LIN {X 0,Y 409.415,Z 604.793,A -85,B 0,C 180,E1 19415.298,E2 19415.298} C_VEL
LIN {X 0,Y 409.395,Z 604.8,A -85,B 0,C 180,E1 19411.55,E2 19411.55} C_VEL
LIN {X 0,Y 409.394,Z 604.798,A -85,B 0,C 180,E1 19407.666,E2 19407.666} C_VEL
LIN {X 0,Y 409.417,Z 604.797,A -85,B 0,C 180,E1 19403.936,E2 19403.936} C_VEL
LIN {X 0,Y 409.444,Z 604.799,A -85,B 0,C 180,E1 19400.041,E2 19400.041} C_VEL
LIN {X 0,Y 409.442,Z 604.791,A -85,B 0,C 180,E1 19396.087,E2 19396.087} C_VEL
LIN {X 0,Y 409.455,Z 604.99,A -85,B 0,C 180,E1 19392.185,E2 19392.185} C_VEL
LIN {X 0,Y 416.656,Z 624.819,A -85,B 0,C 180,E1 19389.076,E2 19389.076} C_VEL
LIN {X 0,Y 424.364,Z 647.273,A -85,B 0,C 180,E1 19385.922,E2 19385.922} C_VEL
LIN {X 0,Y 424.911,Z 649.682,A -85,B 0,C 180,E1 19385.62,E2 19385.62} C_VEL
LIN {X 0,Y 420.58,Z 693.435,A -85,B 0,C 180,E1 19381.336,E2 19381.336} C_VEL
LIN {X 0,Y 423.293,Z 718.927,A -85,B 0,C 180,E1 19380.669,E2 19380.669} C_VEL
LIN {X 0,Y 420.432,Z 893.062,A -85,B 0,C 180,E1 19377.697,E2 19377.697} C_VEL
LIN {X 0,Y 419.51,Z 911.823,A -85,B 0,C 180,E1 19377.138,E2 19377.138} C_VEL
LIN {X 0,Y 418.324,Z 929.671,A -85,B 0,C 180,E1 19376.358,E2 19376.358} C_VEL
LIN {X 0,Y 416.943,Z 947.056,A -85,B 0,C 180,E1 19375.337,E2 19375.337} C_VEL
LIN {X 0,Y 415.337,Z 964.706,A -85,B 0,C 180,E1 19374.007,E2 19374.007} C_VEL
LIN {X 0,Y 413.794,Z 980.489,A -85,B 0,C 180,E1 19372.525,E2 19372.525} C_VEL
LIN {X 0,Y 412.341,Z 995.458,A -85,B 0,C 180,E1 19370.808,E2 19370.808} C_VEL
LIN {X 0,Y 411.026,Z 1009.443,A -85,B 0,C 180,E1 19368.866,E2 19368.866} C_VEL
LIN {X 0,Y 409.929,Z 1022.117,A -85,B 0,C 180,E1 19366.727,E2 19366.727} C_VEL
LIN {X 0,Y 409.153,Z 1033.229,A -85,B 0,C 180,E1 19364.434,E2 19364.434} C_VEL
LIN {X 0,Y 408.687,Z 1042.25,A -85,B 0,C 180,E1 19362.146,E2 19362.146} C_VEL
LIN {X 0,Y 408.488,Z 1049.838,A -85,B 0,C 180,E1 19359.724,E2 19359.724} C_VEL
LIN {X 0,Y 408.479,Z 1055.589,A -85,B 0,C 180,E1 19357.313,E2 19357.313} C_VEL
LIN {X 0,Y 408.559,Z 1059.642,A -85,B 0,C 180,E1 19354.914,E2 19354.914} C_VEL
LIN {X 0,Y 408.661,Z 1062.08,A -85,B 0,C 180,E1 19352.524,E2 19352.524} C_VEL
LIN {X 0,Y 408.725,Z 1062.933,A -85,B 0,C 180,E1 19350,E2 19350} C_VEL
LIN {X 0,Y 408.668,Z 1062.03,A -85,B 0,C 180,E1 19347.476,E2 19347.476} C_VEL
LIN {X 0,Y 408.564,Z 1059.37,A -85,B 0,C 180,E1 19344.946,E2 19344.946} C_VEL
LIN {X 0,Y 408.484,Z 1054.907,A -85,B 0,C 180,E1 19342.405,E2 19342.405} C_VEL
LIN {X 0,Y 408.514,Z 1048.531,A -85,B 0,C 180,E1 19339.85,E2 19339.85} C_VEL
LIN {X 0,Y 408.758,Z 1040.58,A -85,B 0,C 180,E1 19337.419,E2 19337.419} C_VEL
LIN {X 0,Y 409.269,Z 1031.268,A -85,B 0,C 180,E1 19335.137,E2 19335.137} C_VEL
LIN {X 0,Y 410.115,Z 1019.776,A -85,B 0,C 180,E1 19332.843,E2 19332.843} C_VEL
LIN {X 0,Y 411.249,Z 1007.148,A -85,B 0,C 180,E1 19330.765,E2 19330.765} C_VEL
LIN {X 0,Y 412.638,Z 992.973,A -85,B 0,C 180,E1 19328.836,E2 19328.836} C_VEL
LIN {X 0,Y 414.238,Z 977.091,A -85,B 0,C 180,E1 19327.057,E2 19327.057} C_VEL
LIN {X 0,Y 415.901,Z 960.831,A -85,B 0,C 180,E1 19325.575,E2 19325.575} C_VEL
LIN {X 0,Y 417.509,Z 943.547,A -85,B 0,C 180,E1 19324.313,E2 19324.313} C_VEL
LIN {X 0,Y 418.963,Z 925.915,A -85,B 0,C 180,E1 19323.315,E2 19323.315} C_VEL
LIN {X 0,Y 420.212,Z 907.373,A -85,B 0,C 180,E1 19322.551,E2 19322.551} C_VEL
LIN {X 0,Y 421.062,Z 888.73,A -85,B 0,C 180,E1 19322.043,E2 19322.043} C_VEL
LIN {X 0,Y 423.931,Z 716.146,A -85,B 0,C 180,E1 19319.049,E2 19319.049} C_VEL
LIN {X 0,Y 421.384,Z 693.883,A -85,B 0,C 180,E1 19318.403,E2 19318.403} C_VEL
LIN {X 0,Y 426.24,Z 650.86,A -85,B 0,C 180,E1 19314.066,E2 19314.066} C_VEL
LIN {X 0,Y 421.233,Z 635.297,A -85,B 0,C 180,E1 19311.719,E2 19311.719} C_VEL
LIN {X 0,Y 415.789,Z 620.626,A -85,B 0,C 180,E1 19309.243,E2 19309.243} C_VEL
LIN {X 0,Y 410.723,Z 608.35,A -85,B 0,C 180,E1 19306.913,E2 19306.913} C_VEL
LIN {X 0,Y 409.462,Z 604.966,A -85,B 0,C 180,E1 19306.185,E2 19306.185} C_VEL
LIN {X 0,Y 409.409,Z 604.798,A -85,B 0,C 180,E1 19302.38,E2 19302.38} C_VEL
LIN {X 0,Y 409.385,Z 604.791,A -85,B 0,C 180,E1 19298.7,E2 19298.7} C_VEL
LIN {X 0,Y 409.392,Z 604.791,A -85,B 0,C 180,E1 19294.854,E2 19294.854} C_VEL
LIN {X 0,Y 409.423,Z 604.786,A -85,B 0,C 180,E1 19291.18,E2 19291.18} C_VEL
LIN {X 0,Y 409.443,Z 604.781,A -85,B 0,C 180,E1 19287.329,E2 19287.329} C_VEL
LIN {X 0,Y 409.427,Z 604.781,A -85,B 0,C 180,E1 19283.457,E2 19283.457} C_VEL
LIN {X 0,Y 409.402,Z 604.787,A -85,B 0,C 180,E1 19279.696,E2 19279.696} C_VEL
LIN {X 0,Y 409.395,Z 604.797,A -85,B 0,C 180,E1 19275.875,E2 19275.875} C_VEL
LIN {X 0,Y 409.4,Z 604.801,A -85,B 0,C 180,E1 19271.981,E2 19271.981} C_VEL
LIN {X 0,Y 409.417,Z 604.789,A -85,B 0,C 180,E1 19268.143,E2 19268.143} C_VEL
LIN {X 0,Y 409.435,Z 604.778,A -85,B 0,C 180,E1 19264.341,E2 19264.341} C_VEL
LIN {X 0,Y 409.443,Z 604.781,A -85,B 0,C 180,E1 19260.419,E2 19260.419} C_VEL
LIN {X 0,Y 409.424,Z 604.794,A -85,B 0,C 180,E1 19256.499,E2 19256.499} C_VEL
LIN {X 0,Y 409.408,Z 604.799,A -85,B 0,C 180,E1 19252.704,E2 19252.704} C_VEL
LIN {X 0,Y 409.407,Z 604.8,A -85,B 0,C 180,E1 19248.733,E2 19248.733} C_VEL
LIN {X 0,Y 409.408,Z 604.801,A -85,B 0,C 180,E1 19244.725,E2 19244.725} C_VEL
LIN {X 0,Y 409.421,Z 604.8,A -85,B 0,C 180,E1 19240.898,E2 19240.898} C_VEL
LIN {X 0,Y 409.439,Z 604.792,A -85,B 0,C 180,E1 19237,E2 19237} C_VEL
LIN {X 0,Y 409.445,Z 604.787,A -85,B 0,C 180,E1 19232.986,E2 19232.986} C_VEL
LIN {X 0,Y 409.477,Z 605.015,A -85,B 0,C 180,E1 19229.195,E2 19229.195} C_VEL
LIN {X 0,Y 414.075,Z 618.311,A -85,B 0,C 180,E1 19226.096,E2 19226.096} C_VEL
LIN {X 0,Y 418.411,Z 632.268,A -85,B 0,C 180,E1 19223.144,E2 19223.144} C_VEL
LIN {X 0,Y 421.571,Z 644.812,A -85,B 0,C 180,E1 19220.709,E2 19220.709} C_VEL
LIN {X 0,Y 418.574,Z 672.307,A -85,B 0,C 180,E1 19216.567,E2 19216.567} C_VEL
LIN {X 0,Y 415.962,Z 700.171,A -85,B 0,C 180,E1 19212.443,E2 19212.443} C_VEL
LIN {X 0,Y 415.414,Z 707.768,A -85,B 0,C 180,E1 19211.384,E2 19211.384} C_VEL
LIN {X 0,Y 420.157,Z 732.939,A -85,B 0,C 180,E1 19210.505,E2 19210.505} C_VEL
LIN {X 0,Y 418.107,Z 830.68,A -85,B 0,C 180,E1 19208.658,E2 19208.658} C_VEL
LIN {X 0,Y 417.55,Z 846.98,A -85,B 0,C 180,E1 19208.08,E2 19208.08} C_VEL
LIN {X 0,Y 416.769,Z 861.253,A -85,B 0,C 180,E1 19207.317,E2 19207.317} C_VEL
LIN {X 0,Y 415.733,Z 875.611,A -85,B 0,C 180,E1 19206.274,E2 19206.274} C_VEL
LIN {X 0,Y 414.577,Z 888.557,A -85,B 0,C 180,E1 19205.029,E2 19205.029} C_VEL
LIN {X 0,Y 413.441,Z 900.019,A -85,B 0,C 180,E1 19203.629,E2 19203.629} C_VEL
LIN {X 0,Y 412.248,Z 911.043,A -85,B 0,C 180,E1 19201.909,E2 19201.909} C_VEL
LIN {X 0,Y 411.279,Z 919.508,A -85,B 0,C 180,E1 19200.214,E2 19200.214} C_VEL
LIN {X 0,Y 410.461,Z 926.728,A -85,B 0,C 180,E1 19198.36,E2 19198.36} C_VEL
LIN {X 0,Y 409.834,Z 932.478,A -85,B 0,C 180,E1 19196.36,E2 19196.36} C_VEL
LIN {X 0,Y 409.412,Z 936.698,A -85,B 0,C 180,E1 19194.223,E2 19194.223} C_VEL
LIN {X 0,Y 409.166,Z 939.127,A -85,B 0,C 180,E1 19191.955,E2 19191.955} C_VEL
LIN {X 0,Y 409.084,Z 939.659,A -85,B 0,C 180,E1 19189.779,E2 19189.779} C_VEL
LIN {X 0,Y 409.082,Z 939.537,A -85,B 0,C 180,E1 19189.241,E2 19189.241} C_VEL
LIN {X 0,Y 408.111,Z 939.093,A -85,B 0,C 180,E1 19188.162,E2 19188.162} C_VEL
LIN {X 0,Y 403.994,Z 937.675,A -85,B 0,C 180,E1 19186.285,E2 19186.285} C_VEL
LIN {X 0,Y 401.746,Z 935.756,A -85,B 0,C 180,E1 19184.919,E2 19184.919} C_VEL
LIN {X 0,Y 401.569,Z 934.669,A -85,B 0,C 180,E1 19184.384,E2 19184.384} C_VEL
LIN {X 0,Y 402.038,Z 929.349,A -85,B 0,C 180,E1 19182.35,E2 19182.35} C_VEL
LIN {X 0,Y 402.753,Z 921.963,A -85,B 0,C 180,E1 19180.296,E2 19180.296} C_VEL
LIN {X 0,Y 403.589,Z 913.727,A -85,B 0,C 180,E1 19178.548,E2 19178.548} C_VEL
LIN {X 0,Y 404.638,Z 903.344,A -85,B 0,C 180,E1 19176.812,E2 19176.812} C_VEL
LIN {X 0,Y 405.741,Z 891.203,A -85,B 0,C 180,E1 19175.231,E2 19175.231} C_VEL
LIN {X 0,Y 406.821,Z 878.561,A -85,B 0,C 180,E1 19173.946,E2 19173.946} C_VEL
LIN {X 0,Y 407.794,Z 865.03,A -85,B 0,C 180,E1 19172.881,E2 19172.881} C_VEL
LIN {X 0,Y 408.6,Z 850.501,A -85,B 0,C 180,E1 19172.033,E2 19172.033} C_VEL
LIN {X 0,Y 409.183,Z 835.057,A -85,B 0,C 180,E1 19171.41,E2 19171.41} C_VEL
LIN {X 0,Y 409.575,Z 814.247,A -85,B 0,C 180,E1 19170.942,E2 19170.942} C_VEL
LIN {X 0,Y 410.942,Z 731.935,A -85,B 0,C 180,E1 19169.426,E2 19169.426} C_VEL
LIN {X 0,Y 406.656,Z 707.352,A -85,B 0,C 180,E1 19168.661,E2 19168.661} C_VEL
LIN {X 0,Y 409.009,Z 677.997,A -85,B 0,C 180,E1 19164.388,E2 19164.388} C_VEL
LIN {X 0,Y 411.552,Z 650.681,A -85,B 0,C 180,E1 19160.349,E2 19160.349} C_VEL
LIN {X 0,Y 412.189,Z 643.268,A -85,B 0,C 180,E1 19159.235,E2 19159.235} C_VEL
LIN {X 0,Y 407.405,Z 625.4,A -85,B 0,C 180,E1 19155.938,E2 19155.938} C_VEL
LIN {X 0,Y 402.302,Z 608.499,A -85,B 0,C 180,E1 19152.627,E2 19152.627} C_VEL
LIN {X 0,Y 401.507,Z 605.885,A -85,B 0,C 180,E1 19152.013,E2 19152.013} C_VEL
LIN {X 0,Y 401.5,Z 605.772,A -85,B 0,C 180,E1 19148.065,E2 19148.065} C_VEL
LIN {X 0,Y 401.498,Z 605.771,A -85,B 0,C 180,E1 19144.004,E2 19144.004} C_VEL
LIN {X 0,Y 401.499,Z 605.737,A -85,B 0,C 180,E1 19140.07,E2 19140.07} C_VEL
LIN {X 0,Y 401.502,Z 605.778,A -85,B 0,C 180,E1 19136.024,E2 19136.024} C_VEL
LIN {X 0,Y 401.502,Z 605.772,A -85,B 0,C 180,E1 19132.04,E2 19132.04} C_VEL
LIN {X 0,Y 401.498,Z 605.772,A -85,B 0,C 180,E1 19128.126,E2 19128.126} C_VEL
LIN {X 0,Y 401.491,Z 605.787,A -85,B 0,C 180,E1 19124.173,E2 19124.173} C_VEL
LIN {X 0,Y 401.477,Z 605.762,A -85,B 0,C 180,E1 19120.351,E2 19120.351} C_VEL
LIN {X 0,Y 401.478,Z 605.785,A -85,B 0,C 180,E1 19116.351,E2 19116.351} C_VEL
LIN {X 0,Y 401.479,Z 605.771,A -85,B 0,C 180,E1 19112.374,E2 19112.374} C_VEL
LIN {X 0,Y 401.495,Z 605.778,A -85,B 0,C 180,E1 19108.466,E2 19108.466} C_VEL
LIN {X 0,Y 401.499,Z 605.765,A -85,B 0,C 180,E1 19104.575,E2 19104.575} C_VEL
LIN {X 0,Y 401.506,Z 605.779,A -85,B 0,C 180,E1 19100.709,E2 19100.709} C_VEL
LIN {X 0,Y 401.492,Z 605.755,A -85,B 0,C 180,E1 19096.791,E2 19096.791} C_VEL
LIN {X 0,Y 401.476,Z 605.789,A -85,B 0,C 180,E1 19092.953,E2 19092.953} C_VEL
LIN {X 0,Y 401.464,Z 605.755,A -85,B 0,C 180,E1 19089.028,E2 19089.028} C_VEL
LIN {X 0,Y 401.468,Z 605.784,A -85,B 0,C 180,E1 19085.144,E2 19085.144} C_VEL
LIN {X 0,Y 401.474,Z 605.759,A -85,B 0,C 180,E1 19081.285,E2 19081.285} C_VEL
LIN {X 0,Y 401.495,Z 605.783,A -85,B 0,C 180,E1 19077.431,E2 19077.431} C_VEL
LIN {X 0,Y 401.509,Z 605.756,A -85,B 0,C 180,E1 19073.423,E2 19073.423} C_VEL
LIN {X 0,Y 401.503,Z 605.786,A -85,B 0,C 180,E1 19069.381,E2 19069.381} C_VEL
LIN {X 0,Y 401.501,Z 605.762,A -85,B 0,C 180,E1 19065.433,E2 19065.433} C_VEL
LIN {X 0,Y 401.477,Z 605.788,A -85,B 0,C 180,E1 19061.562,E2 19061.562} C_VEL
LIN {X 0,Y 401.453,Z 605.782,A -85,B 0,C 180,E1 19057.755,E2 19057.755} C_VEL
LIN {X 0,Y 401.456,Z 605.772,A -85,B 0,C 180,E1 19053.843,E2 19053.843} C_VEL
LIN {X 0,Y 401.471,Z 605.781,A -85,B 0,C 180,E1 19050.077,E2 19050.077} C_VEL
LIN {X 0,Y 401.494,Z 605.781,A -85,B 0,C 180,E1 19046.266,E2 19046.266} C_VEL
LIN {X 0,Y 401.506,Z 605.78,A -85,B 0,C 180,E1 19042.365,E2 19042.365} C_VEL
LIN {X 0,Y 401.484,Z 605.78,A -85,B 0,C 180,E1 19038.513,E2 19038.513} C_VEL
LIN {X 0,Y 401.455,Z 605.786,A -85,B 0,C 180,E1 19034.78,E2 19034.78} C_VEL
LIN {X 0,Y 401.487,Z 606.048,A -85,B 0,C 180,E1 19032.879,E2 19032.879} C_VEL
LIN {X 0,Y 408.321,Z 624.696,A -85,B 0,C 180,E1 19029.866,E2 19029.866} C_VEL
LIN {X 0,Y 415.634,Z 645.93,A -85,B 0,C 180,E1 19026.768,E2 19026.768} C_VEL
LIN {X 0,Y 417.528,Z 652.187,A -85,B 0,C 180,E1 19025.924,E2 19025.924} C_VEL
LIN {X 0,Y 413.207,Z 693.553,A -85,B 0,C 180,E1 19021.797,E2 19021.797} C_VEL
LIN {X 0,Y 415.955,Z 719.877,A -85,B 0,C 180,E1 19021.094,E2 19021.094} C_VEL
LIN {X 0,Y 412.963,Z 892.44,A -85,B 0,C 180,E1 19018.099,E2 19018.099} C_VEL
LIN {X 0,Y 412.015,Z 911.066,A -85,B 0,C 180,E1 19017.536,E2 19017.536} C_VEL
LIN {X 0,Y 410.749,Z 929.303,A -85,B 0,C 180,E1 19016.723,E2 19016.723} C_VEL
LIN {X 0,Y 409.229,Z 947.539,A -85,B 0,C 180,E1 19015.624,E2 19015.624} C_VEL
LIN {X 0,Y 407.642,Z 964.222,A -85,B 0,C 180,E1 19014.335,E2 19014.335} C_VEL
LIN {X 0,Y 406.038,Z 979.927,A -85,B 0,C 180,E1 19012.831,E2 19012.831} C_VEL
LIN {X 0,Y 404.516,Z 994.883,A -85,B 0,C 180,E1 19011.078,E2 19011.078} C_VEL
LIN {X 0,Y 403.141,Z 1008.778,A -85,B 0,C 180,E1 19009.101,E2 19009.101} C_VEL
LIN {X 0,Y 401.998,Z 1021.371,A -85,B 0,C 180,E1 19006.919,E2 19006.919} C_VEL
LIN {X 0,Y 401.192,Z 1032.422,A -85,B 0,C 180,E1 19004.579,E2 19004.579} C_VEL
LIN {X 0,Y 400.719,Z 1041.383,A -85,B 0,C 180,E1 19002.245,E2 19002.245} C_VEL
LIN {X 0,Y 400.525,Z 1048.91,A -85,B 0,C 180,E1 18999.774,E2 18999.774} C_VEL
LIN {X 0,Y 400.535,Z 1054.603,A -85,B 0,C 180,E1 18997.315,E2 18997.315} C_VEL
LIN {X 0,Y 400.634,Z 1058.591,A -85,B 0,C 180,E1 18994.868,E2 18994.868} C_VEL
LIN {X 0,Y 400.752,Z 1060.959,A -85,B 0,C 180,E1 18992.431,E2 18992.431} C_VEL
LIN {X 0,Y 400.814,Z 1061.738,A -85,B 0,C 180,E1 18990,E2 18990} C_VEL
LIN {X 0,Y 400.749,Z 1060.835,A -85,B 0,C 180,E1 18987.426,E2 18987.426} C_VEL
LIN {X 0,Y 400.628,Z 1058.172,A -85,B 0,C 180,E1 18984.845,E2 18984.845} C_VEL
LIN {X 0,Y 400.524,Z 1053.7,A -85,B 0,C 180,E1 18982.253,E2 18982.253} C_VEL
LIN {X 0,Y 400.547,Z 1047.303,A -85,B 0,C 180,E1 18979.646,E2 18979.646} C_VEL
LIN {X 0,Y 400.805,Z 1039.353,A -85,B 0,C 180,E1 18977.172,E2 18977.172} C_VEL
LIN {X 0,Y 401.352,Z 1029.981,A -85,B 0,C 180,E1 18974.836,E2 18974.836} C_VEL
LIN {X 0,Y 402.191,Z 1019.26,A -85,B 0,C 180,E1 18972.643,E2 18972.643} C_VEL
LIN {X 0,Y 403.427,Z 1006.277,A -85,B 0,C 180,E1 18970.453,E2 18970.453} C_VEL
LIN {X 0,Y 404.899,Z 992.192,A -85,B 0,C 180,E1 18968.488,E2 18968.488} C_VEL
LIN {X 0,Y 406.594,Z 976.399,A -85,B 0,C 180,E1 18966.677,E2 18966.677} C_VEL
LIN {X 0,Y 408.354,Z 960.2,A -85,B 0,C 180,E1 18965.171,E2 18965.171} C_VEL
LIN {X 0,Y 410.046,Z 942.983,A -85,B 0,C 180,E1 18963.888,E2 18963.888} C_VEL
LIN {X 0,Y 411.554,Z 925.702,A -85,B 0,C 180,E1 18962.889,E2 18962.889} C_VEL
LIN {X 0,Y 412.893,Z 907.092,A -85,B 0,C 180,E1 18962.101,E2 18962.101} C_VEL
LIN {X 0,Y 413.796,Z 888.177,A -85,B 0,C 180,E1 18961.575,E2 18961.575} C_VEL
LIN {X 0,Y 416.851,Z 717.196,A -85,B 0,C 180,E1 18958.556,E2 18958.556} C_VEL
LIN {X 0,Y 414.253,Z 694.007,A -85,B 0,C 180,E1 18957.859,E2 18957.859} C_VEL
LIN {X 0,Y 419.097,Z 653.502,A -85,B 0,C 180,E1 18953.682,E2 18953.682} C_VEL
LIN {X 0,Y 414.062,Z 637.9,A -85,B 0,C 180,E1 18951.257,E2 18951.257} C_VEL
LIN {X 0,Y 408.413,Z 622.902,A -85,B 0,C 180,E1 18948.624,E2 18948.624} C_VEL
LIN {X 0,Y 403.938,Z 612.2,A -85,B 0,C 180,E1 18946.518,E2 18946.518} C_VEL
LIN {X 0,Y 401.475,Z 605.966,A -85,B 0,C 180,E1 18945.16,E2 18945.16} C_VEL
LIN {X 0,Y 401.47,Z 605.78,A -85,B 0,C 180,E1 18941.441,E2 18941.441} C_VEL
LIN {X 0,Y 401.503,Z 605.777,A -85,B 0,C 180,E1 18937.635,E2 18937.635} C_VEL
LIN {X 0,Y 401.495,Z 605.785,A -85,B 0,C 180,E1 18933.719,E2 18933.719} C_VEL
LIN {X 0,Y 401.476,Z 605.788,A -85,B 0,C 180,E1 18929.874,E2 18929.874} C_VEL
LIN {X 0,Y 401.462,Z 605.789,A -85,B 0,C 180,E1 18925.998,E2 18925.998} C_VEL
LIN {X 0,Y 401.453,Z 605.787,A -85,B 0,C 180,E1 18922.091,E2 18922.091} C_VEL
LIN {X 0,Y 401.456,Z 605.777,A -85,B 0,C 180,E1 18918.139,E2 18918.139} C_VEL
LIN {X 0,Y 401.466,Z 605.77,A -85,B 0,C 180,E1 18914.274,E2 18914.274} C_VEL
LIN {X 0,Y 401.493,Z 605.772,A -85,B 0,C 180,E1 18910.474,E2 18910.474} C_VEL
LIN {X 0,Y 401.509,Z 605.783,A -85,B 0,C 180,E1 18906.479,E2 18906.479} C_VEL
LIN {X 0,Y 401.5,Z 605.784,A -85,B 0,C 180,E1 18902.426,E2 18902.426} C_VEL
LIN {X 0,Y 401.487,Z 605.778,A -85,B 0,C 180,E1 18898.573,E2 18898.573} C_VEL
LIN {X 0,Y 401.469,Z 605.771,A -85,B 0,C 180,E1 18894.712,E2 18894.712} C_VEL
LIN {X 0,Y 401.465,Z 605.77,A -85,B 0,C 180,E1 18890.828,E2 18890.828} C_VEL
LIN {X 0,Y 401.468,Z 605.772,A -85,B 0,C 180,E1 18886.853,E2 18886.853} C_VEL
LIN {X 0,Y 401.482,Z 605.774,A -85,B 0,C 180,E1 18883.004,E2 18883.004} C_VEL
LIN {X 0,Y 401.498,Z 605.774,A -85,B 0,C 180,E1 18879.046,E2 18879.046} C_VEL
LIN {X 0,Y 401.502,Z 605.779,A -85,B 0,C 180,E1 18875.111,E2 18875.111} C_VEL
LIN {X 0,Y 401.507,Z 605.779,A -85,B 0,C 180,E1 18871.111,E2 18871.111} C_VEL
LIN {X 0,Y 401.524,Z 606.105,A -85,B 0,C 180,E1 18870.156,E2 18870.156} C_VEL
LIN {X 0,Y 406.115,Z 618.877,A -85,B 0,C 180,E1 18867.036,E2 18867.036} C_VEL
LIN {X 0,Y 410.65,Z 633.112,A -85,B 0,C 180,E1 18863.897,E2 18863.897} C_VEL
LIN {X 0,Y 414.322,Z 647.351,A -85,B 0,C 180,E1 18861.04,E2 18861.04} C_VEL
LIN {X 0,Y 411.328,Z 673.554,A -85,B 0,C 180,E1 18857.027,E2 18857.027} C_VEL
LIN {X 0,Y 408.488,Z 701.978,A -85,B 0,C 180,E1 18852.75,E2 18852.75} C_VEL
LIN {X 0,Y 408.062,Z 707.405,A -85,B 0,C 180,E1 18851.984,E2 18851.984} C_VEL
LIN {X 0,Y 413.061,Z 733.503,A -85,B 0,C 180,E1 18851.027,E2 18851.027} C_VEL
LIN {X 0,Y 410.923,Z 831.377,A -85,B 0,C 180,E1 18849.136,E2 18849.136} C_VEL
LIN {X 0,Y 410.326,Z 847.718,A -85,B 0,C 180,E1 18848.545,E2 18848.545} C_VEL
LIN {X 0,Y 409.469,Z 862.358,A -85,B 0,C 180,E1 18847.745,E2 18847.745} C_VEL
LIN {X 0,Y 408.369,Z 876.626,A -85,B 0,C 180,E1 18846.685,E2 18846.685} C_VEL
LIN {X 0,Y 407.094,Z 889.994,A -85,B 0,C 180,E1 18845.37,E2 18845.37} C_VEL
LIN {X 0,Y 405.926,Z 901.003,A -85,B 0,C 180,E1 18843.996,E2 18843.996} C_VEL
LIN {X 0,Y 404.656,Z 911.975,A -85,B 0,C 180,E1 18842.256,E2 18842.256} C_VEL
LIN {X 0,Y 403.556,Z 920.904,A -85,B 0,C 180,E1 18840.433,E2 18840.433} C_VEL
LIN {X 0,Y 402.653,Z 928.312,A -85,B 0,C 180,E1 18838.472,E2 18838.472} C_VEL
LIN {X 0,Y 401.942,Z 934.289,A -85,B 0,C 180,E1 18836.282,E2 18836.282} C_VEL
LIN {X 0,Y 401.527,Z 938.036,A -85,B 0,C 180,E1 18834.26,E2 18834.26} C_VEL
LIN {X 0,Y 401.263,Z 940.392,A -85,B 0,C 180,E1 18831.948,E2 18831.948} C_VEL
LIN {X 0,Y 401.175,Z 940.858,A -85,B 0,C 180,E1 18829.813,E2 18829.813} C_VEL
LIN {X 0,Y 401.22,Z 939.617,A -85,B 0,C 180,E1 18827.55,E2 18827.55} C_VEL
LIN {X 0,Y 401.424,Z 936.51,A -85,B 0,C 180,E1 18825.309,E2 18825.309} C_VEL
LIN {X 0,Y 401.569,Z 934.669,A -85,B 0,C 180,E1 18824.384,E2 18824.384} C_VEL
LIN {X 0,Y 400.81,Z 932.367,A -85,B 0,C 180,E1 18823.329,E2 18823.329} C_VEL
LIN {X 0,Y 397.259,Z 927.986,A -85,B 0,C 180,E1 18821.577,E2 18821.577} C_VEL
LIN {X 0,Y 395.218,Z 923.781,A -85,B 0,C 180,E1 18820.292,E2 18820.292} C_VEL
LIN {X 0,Y 395.106,Z 921.534,A -85,B 0,C 180,E1 18819.737,E2 18819.737} C_VEL
LIN {X 0,Y 396.111,Z 912.264,A -85,B 0,C 180,E1 18817.834,E2 18817.834} C_VEL
LIN {X 0,Y 397.261,Z 901.138,A -85,B 0,C 180,E1 18816.068,E2 18816.068} C_VEL
LIN {X 0,Y 398.363,Z 889.461,A -85,B 0,C 180,E1 18814.607,E2 18814.607} C_VEL
LIN {X 0,Y 399.538,Z 876.086,A -85,B 0,C 180,E1 18813.299,E2 18813.299} C_VEL
LIN {X 0,Y 400.493,Z 862.539,A -85,B 0,C 180,E1 18812.289,E2 18812.289} C_VEL
LIN {X 0,Y 401.315,Z 847.48,A -85,B 0,C 180,E1 18811.459,E2 18811.459} C_VEL
LIN {X 0,Y 401.873,Z 830.698,A -85,B 0,C 180,E1 18810.855,E2 18810.855} C_VEL
LIN {X 0,Y 403.57,Z 732.835,A -85,B 0,C 180,E1 18808.984,E2 18808.984} C_VEL
LIN {X 0,Y 399.109,Z 707.145,A -85,B 0,C 180,E1 18808.169,E2 18808.169} C_VEL
LIN {X 0,Y 401.601,Z 677.995,A -85,B 0,C 180,E1 18803.854,E2 18803.854} C_VEL
LIN {X 0,Y 404.312,Z 650.623,A -85,B 0,C 180,E1 18799.743,E2 18799.743} C_VEL
LIN {X 0,Y 404.772,Z 645.971,A -85,B 0,C 180,E1 18799.035,E2 18799.035} C_VEL
LIN {X 0,Y 400.003,Z 628.055,A -85,B 0,C 180,E1 18795.672,E2 18795.672} C_VEL
LIN {X 0,Y 395.016,Z 611.616,A -85,B 0,C 180,E1 18792.393,E2 18792.393} C_VEL
LIN {X 0,Y 393.571,Z 606.878,A -85,B 0,C 180,E1 18791.331,E2 18791.331} C_VEL
LIN {X 0,Y 393.55,Z 606.741,A -85,B 0,C 180,E1 18787.283,E2 18787.283} C_VEL
LIN {X 0,Y 393.55,Z 606.774,A -85,B 0,C 180,E1 18783.276,E2 18783.276} C_VEL
LIN {X 0,Y 393.539,Z 606.719,A -85,B 0,C 180,E1 18779.291,E2 18779.291} C_VEL
LIN {X 0,Y 393.55,Z 606.774,A -85,B 0,C 180,E1 18775.312,E2 18775.312} C_VEL
LIN {X 0,Y 393.553,Z 606.768,A -85,B 0,C 180,E1 18771.258,E2 18771.258} C_VEL
LIN {X 0,Y 393.559,Z 606.753,A -85,B 0,C 180,E1 18767.457,E2 18767.457} C_VEL
LIN {X 0,Y 393.563,Z 606.77,A -85,B 0,C 180,E1 18763.398,E2 18763.398} C_VEL
LIN {X 0,Y 393.565,Z 606.759,A -85,B 0,C 180,E1 18759.43,E2 18759.43} C_VEL
LIN {X 0,Y 393.559,Z 606.758,A -85,B 0,C 180,E1 18755.398,E2 18755.398} C_VEL
LIN {X 0,Y 393.561,Z 606.767,A -85,B 0,C 180,E1 18751.387,E2 18751.387} C_VEL
LIN {X 0,Y 393.542,Z 606.757,A -85,B 0,C 180,E1 18747.538,E2 18747.538} C_VEL
LIN {X 0,Y 393.532,Z 606.765,A -85,B 0,C 180,E1 18743.668,E2 18743.668} C_VEL
LIN {X 0,Y 393.535,Z 606.768,A -85,B 0,C 180,E1 18739.75,E2 18739.75} C_VEL
LIN {X 0,Y 393.537,Z 606.76,A -85,B 0,C 180,E1 18735.775,E2 18735.775} C_VEL
LIN {X 0,Y 393.551,Z 606.767,A -85,B 0,C 180,E1 18731.876,E2 18731.876} C_VEL
LIN {X 0,Y 393.565,Z 606.745,A -85,B 0,C 180,E1 18727.885,E2 18727.885} C_VEL
LIN {X 0,Y 393.562,Z 606.768,A -85,B 0,C 180,E1 18723.934,E2 18723.934} C_VEL
LIN {X 0,Y 393.57,Z 606.743,A -85,B 0,C 180,E1 18719.855,E2 18719.855} C_VEL
LIN {X 0,Y 393.561,Z 606.771,A -85,B 0,C 180,E1 18715.775,E2 18715.775} C_VEL
LIN {X 0,Y 393.55,Z 606.749,A -85,B 0,C 180,E1 18711.821,E2 18711.821} C_VEL
LIN {X 0,Y 393.528,Z 606.777,A -85,B 0,C 180,E1 18707.975,E2 18707.975} C_VEL
LIN {X 0,Y 393.518,Z 606.766,A -85,B 0,C 180,E1 18704.073,E2 18704.073} C_VEL
LIN {X 0,Y 393.521,Z 606.764,A -85,B 0,C 180,E1 18700.07,E2 18700.07} C_VEL
LIN {X 0,Y 393.526,Z 606.776,A -85,B 0,C 180,E1 18696.161,E2 18696.161} C_VEL
LIN {X 0,Y 393.545,Z 606.774,A -85,B 0,C 180,E1 18692.294,E2 18692.294} C_VEL
LIN {X 0,Y 393.564,Z 606.762,A -85,B 0,C 180,E1 18688.443,E2 18688.443} C_VEL
LIN {X 0,Y 393.562,Z 606.765,A -85,B 0,C 180,E1 18684.388,E2 18684.388} C_VEL
LIN {X 0,Y 393.57,Z 606.77,A -85,B 0,C 180,E1 18680.334,E2 18680.334} C_VEL
LIN {X 0,Y 393.555,Z 606.771,A -85,B 0,C 180,E1 18676.288,E2 18676.288} C_VEL
LIN {X 0,Y 393.587,Z 607.064,A -85,B 0,C 180,E1 18673.614,E2 18673.614} C_VEL
LIN {X 0,Y 400.611,Z 626.198,A -85,B 0,C 180,E1 18670.428,E2 18670.428} C_VEL
LIN {X 0,Y 407.631,Z 646.517,A -85,B 0,C 180,E1 18667.371,E2 18667.371} C_VEL
LIN {X 0,Y 410.135,Z 654.695,A -85,B 0,C 180,E1 18666.233,E2 18666.233} C_VEL
LIN {X 0,Y 405.844,Z 694.221,A -85,B 0,C 180,E1 18662.235,E2 18662.235} C_VEL
LIN {X 0,Y 408.638,Z 720.771,A -85,B 0,C 180,E1 18661.535,E2 18661.535} C_VEL
LIN {X 0,Y 405.518,Z 891.82,A -85,B 0,C 180,E1 18658.517,E2 18658.517} C_VEL
LIN {X 0,Y 404.532,Z 910.424,A -85,B 0,C 180,E1 18657.944,E2 18657.944} C_VEL
LIN {X 0,Y 403.258,Z 928.162,A -85,B 0,C 180,E1 18657.144,E2 18657.144} C_VEL
LIN {X 0,Y 401.695,Z 946.088,A -85,B 0,C 180,E1 18656.053,E2 18656.053} C_VEL
LIN {X 0,Y 400.049,Z 962.797,A -85,B 0,C 180,E1 18654.749,E2 18654.749} C_VEL
LIN {X 0,Y 398.349,Z 978.685,A -85,B 0,C 180,E1 18653.208,E2 18653.208} C_VEL
LIN {X 0,Y 396.759,Z 993.634,A -85,B 0,C 180,E1 18651.433,E2 18651.433} C_VEL
LIN {X 0,Y 395.357,Z 1007.064,A -85,B 0,C 180,E1 18649.502,E2 18649.502} C_VEL
LIN {X 0,Y 394.137,Z 1019.885,A -85,B 0,C 180,E1 18647.266,E2 18647.266} C_VEL
LIN {X 0,Y 393.273,Z 1031.006,A -85,B 0,C 180,E1 18644.88,E2 18644.88} C_VEL
LIN {X 0,Y 392.771,Z 1040.027,A -85,B 0,C 180,E1 18642.497,E2 18642.497} C_VEL
LIN {X 0,Y 392.563,Z 1047.603,A -85,B 0,C 180,E1 18639.974,E2 18639.974} C_VEL
LIN {X 0,Y 392.584,Z 1053.339,A -85,B 0,C 180,E1 18637.464,E2 18637.464} C_VEL
LIN {X 0,Y 392.702,Z 1057.361,A -85,B 0,C 180,E1 18634.966,E2 18634.966} C_VEL
LIN {X 0,Y 392.834,Z 1059.753,A -85,B 0,C 180,E1 18632.48,E2 18632.48} C_VEL
LIN {X 0,Y 392.899,Z 1060.536,A -85,B 0,C 180,E1 18629.854,E2 18629.854} C_VEL
LIN {X 0,Y 392.822,Z 1059.545,A -85,B 0,C 180,E1 18627.228,E2 18627.228} C_VEL
LIN {X 0,Y 392.678,Z 1056.777,A -85,B 0,C 180,E1 18624.594,E2 18624.594} C_VEL
LIN {X 0,Y 392.563,Z 1052.178,A -85,B 0,C 180,E1 18621.947,E2 18621.947} C_VEL
LIN {X 0,Y 392.581,Z 1046.073,A -85,B 0,C 180,E1 18619.434,E2 18619.434} C_VEL
LIN {X 0,Y 392.857,Z 1038.098,A -85,B 0,C 180,E1 18616.908,E2 18616.908} C_VEL
LIN {X 0,Y 393.44,Z 1028.707,A -85,B 0,C 180,E1 18614.524,E2 18614.524} C_VEL
LIN {X 0,Y 394.347,Z 1017.99,A -85,B 0,C 180,E1 18612.287,E2 18612.287} C_VEL
LIN {X 0,Y 395.569,Z 1005.965,A -85,B 0,C 180,E1 18610.202,E2 18610.202} C_VEL
LIN {X 0,Y 397.113,Z 992.022,A -85,B 0,C 180,E1 18608.2,E2 18608.2} C_VEL
LIN {X 0,Y 398.813,Z 977.089,A -85,B 0,C 180,E1 18606.429,E2 18606.429} C_VEL
LIN {X 0,Y 400.732,Z 960.405,A -85,B 0,C 180,E1 18604.823,E2 18604.823} C_VEL
LIN {X 0,Y 402.48,Z 943.643,A -85,B 0,C 180,E1 18603.532,E2 18603.532} C_VEL
LIN {X 0,Y 404.112,Z 926.099,A -85,B 0,C 180,E1 18602.48,E2 18602.48} C_VEL
LIN {X 0,Y 405.526,Z 907.91,A -85,B 0,C 180,E1 18601.673,E2 18601.673} C_VEL
LIN {X 0,Y 406.542,Z 888.994,A -85,B 0,C 180,E1 18601.112,E2 18601.112} C_VEL
LIN {X 0,Y 409.813,Z 718.116,A -85,B 0,C 180,E1 18598.035,E2 18598.035} C_VEL
LIN {X 0,Y 407.162,Z 694.203,A -85,B 0,C 180,E1 18597.3,E2 18597.3} C_VEL
LIN {X 0,Y 411.934,Z 656.195,A -85,B 0,C 180,E1 18593.289,E2 18593.289} C_VEL
LIN {X 0,Y 407.031,Z 640.971,A -85,B 0,C 180,E1 18590.853,E2 18590.853} C_VEL
LIN {X 0,Y 401.735,Z 626.845,A -85,B 0,C 180,E1 18588.301,E2 18588.301} C_VEL
LIN {X 0,Y 396.571,Z 614.146,A -85,B 0,C 180,E1 18585.728,E2 18585.728} C_VEL
LIN {X 0,Y 393.592,Z 607.031,A -85,B 0,C 180,E1 18584.111,E2 18584.111} C_VEL
LIN {X 0,Y 393.529,Z 606.778,A -85,B 0,C 180,E1 18580.339,E2 18580.339} C_VEL
LIN {X 0,Y 393.516,Z 606.779,A -85,B 0,C 180,E1 18576.481,E2 18576.481} C_VEL
LIN {X 0,Y 393.513,Z 606.771,A -85,B 0,C 180,E1 18572.482,E2 18572.482} C_VEL
LIN {X 0,Y 393.513,Z 606.768,A -85,B 0,C 180,E1 18568.462,E2 18568.462} C_VEL
LIN {X 0,Y 393.521,Z 606.769,A -85,B 0,C 180,E1 18564.549,E2 18564.549} C_VEL
LIN {X 0,Y 393.547,Z 606.773,A -85,B 0,C 180,E1 18560.779,E2 18560.779} C_VEL
LIN {X 0,Y 393.561,Z 606.774,A -85,B 0,C 180,E1 18556.835,E2 18556.835} C_VEL
LIN {X 0,Y 393.559,Z 606.766,A -85,B 0,C 180,E1 18552.918,E2 18552.918} C_VEL
LIN {X 0,Y 393.548,Z 606.754,A -85,B 0,C 180,E1 18548.915,E2 18548.915} C_VEL
LIN {X 0,Y 393.528,Z 606.759,A -85,B 0,C 180,E1 18545.102,E2 18545.102} C_VEL
LIN {X 0,Y 393.524,Z 606.773,A -85,B 0,C 180,E1 18541.164,E2 18541.164} C_VEL
LIN {X 0,Y 393.527,Z 606.777,A -85,B 0,C 180,E1 18537.233,E2 18537.233} C_VEL
LIN {X 0,Y 393.533,Z 606.778,A -85,B 0,C 180,E1 18533.288,E2 18533.288} C_VEL
LIN {X 0,Y 393.551,Z 606.766,A -85,B 0,C 180,E1 18529.46,E2 18529.46} C_VEL
LIN {X 0,Y 393.566,Z 606.764,A -85,B 0,C 180,E1 18525.433,E2 18525.433} C_VEL
LIN {X 0,Y 393.565,Z 606.77,A -85,B 0,C 180,E1 18521.372,E2 18521.372} C_VEL
LIN {X 0,Y 393.571,Z 606.773,A -85,B 0,C 180,E1 18517.284,E2 18517.284} C_VEL
LIN {X 0,Y 393.565,Z 606.765,A -85,B 0,C 180,E1 18513.277,E2 18513.277} C_VEL
LIN {X 0,Y 393.612,Z 607.061,A -85,B 0,C 180,E1 18511.214,E2 18511.214} C_VEL
LIN {X 0,Y 398.188,Z 619.585,A -85,B 0,C 180,E1 18508.006,E2 18508.006} C_VEL
LIN {X 0,Y 402.446,Z 632.731,A -85,B 0,C 180,E1 18504.976,E2 18504.976} C_VEL
LIN {X 0,Y 406.273,Z 646.754,A -85,B 0,C 180,E1 18502.028,E2 18502.028} C_VEL
LIN {X 0,Y 407.034,Z 650.97,A -85,B 0,C 180,E1 18501.215,E2 18501.215} C_VEL
LIN {X 0,Y 403.799,Z 677.583,A -85,B 0,C 180,E1 18497.083,E2 18497.083} C_VEL
LIN {X 0,Y 400.806,Z 706.092,A -85,B 0,C 180,E1 18492.729,E2 18492.729} C_VEL
LIN {X 0,Y 400.944,Z 708.531,A -85,B 0,C 180,E1 18492.515,E2 18492.515} C_VEL
LIN {X 0,Y 406.088,Z 735.18,A -85,B 0,C 180,E1 18491.539,E2 18491.539} C_VEL
LIN {X 0,Y 403.789,Z 832.031,A -85,B 0,C 180,E1 18489.637,E2 18489.637} C_VEL
LIN {X 0,Y 403.16,Z 848.305,A -85,B 0,C 180,E1 18489.039,E2 18489.039} C_VEL
LIN {X 0,Y 402.264,Z 862.87,A -85,B 0,C 180,E1 18488.236,E2 18488.236} C_VEL
LIN {X 0,Y 401.112,Z 877.059,A -85,B 0,C 180,E1 18487.172,E2 18487.172} C_VEL
LIN {X 0,Y 399.784,Z 890.21,A -85,B 0,C 180,E1 18485.872,E2 18485.872} C_VEL
LIN {X 0,Y 398.44,Z 902.058,A -85,B 0,C 180,E1 18484.376,E2 18484.376} C_VEL
LIN {X 0,Y 397.077,Z 913.006,A -85,B 0,C 180,E1 18482.606,E2 18482.606} C_VEL
LIN {X 0,Y 395.945,Z 921.562,A -85,B 0,C 180,E1 18480.839,E2 18480.839} C_VEL
LIN {X 0,Y 394.912,Z 929.351,A -85,B 0,C 180,E1 18478.754,E2 18478.754} C_VEL
LIN {X 0,Y 394.176,Z 935.005,A -85,B 0,C 180,E1 18476.678,E2 18476.678} C_VEL
LIN {X 0,Y 393.671,Z 939.163,A -85,B 0,C 180,E1 18474.456,E2 18474.456} C_VEL
LIN {X 0,Y 393.371,Z 941.549,A -85,B 0,C 180,E1 18472.097,E2 18472.097} C_VEL
LIN {X 0,Y 393.265,Z 942.054,A -85,B 0,C 180,E1 18469.828,E2 18469.828} C_VEL
LIN {X 0,Y 393.314,Z 940.742,A -85,B 0,C 180,E1 18467.456,E2 18467.456} C_VEL
LIN {X 0,Y 393.549,Z 937.456,A -85,B 0,C 180,E1 18465.106,E2 18465.106} C_VEL
LIN {X 0,Y 393.977,Z 932.628,A -85,B 0,C 180,E1 18462.955,E2 18462.955} C_VEL
LIN {X 0,Y 394.658,Z 925.816,A -85,B 0,C 180,E1 18460.805,E2 18460.805} C_VEL
LIN {X 0,Y 395.106,Z 921.534,A -85,B 0,C 180,E1 18459.737,E2 18459.737} C_VEL
LIN {X 0,Y 394.583,Z 917.466,A -85,B 0,C 180,E1 18458.785,E2 18458.785} C_VEL
LIN {X 0,Y 390.934,Z 909.001,A -85,B 0,C 180,E1 18456.944,E2 18456.944} C_VEL
LIN {X 0,Y 389.657,Z 903.305,A -85,B 0,C 180,E1 18455.949,E2 18455.949} C_VEL
LIN {X 0,Y 389.721,Z 900.948,A -85,B 0,C 180,E1 18455.597,E2 18455.597} C_VEL
LIN {X 0,Y 390.933,Z 888.518,A -85,B 0,C 180,E1 18454.067,E2 18454.067} C_VEL
LIN {X 0,Y 392.07,Z 875.937,A -85,B 0,C 180,E1 18452.85,E2 18452.85} C_VEL
LIN {X 0,Y 393.154,Z 860.961,A -85,B 0,C 180,E1 18451.749,E2 18451.749} C_VEL
LIN {X 0,Y 393.949,Z 845.796,A -85,B 0,C 180,E1 18450.949,E2 18450.949} C_VEL
LIN {X 0,Y 394.467,Z 830.15,A -85,B 0,C 180,E1 18450.406,E2 18450.406} C_VEL
LIN {X 0,Y 396.241,Z 734.006,A -85,B 0,C 180,E1 18448.545,E2 18448.545} C_VEL
LIN {X 0,Y 391.588,Z 706.936,A -85,B 0,C 180,E1 18447.658,E2 18447.658} C_VEL
LIN {X 0,Y 394.223,Z 677.972,A -85,B 0,C 180,E1 18443.3,E2 18443.3} C_VEL
LIN {X 0,Y 397.12,Z 650.417,A -85,B 0,C 180,E1 18439.095,E2 18439.095} C_VEL
LIN {X 0,Y 397.147,Z 647.82,A -85,B 0,C 180,E1 18438.675,E2 18438.675} C_VEL
LIN {X 0,Y 392.388,Z 629.909,A -85,B 0,C 180,E1 18435.237,E2 18435.237} C_VEL
LIN {X 0,Y 387.25,Z 613.02,A -85,B 0,C 180,E1 18431.795,E2 18431.795} C_VEL
LIN {X 0,Y 385.635,Z 607.862,A -85,B 0,C 180,E1 18430.617,E2 18430.617} C_VEL
LIN {X 0,Y 385.619,Z 607.718,A -85,B 0,C 180,E1 18426.618,E2 18426.618} C_VEL
LIN {X 0,Y 385.625,Z 607.763,A -85,B 0,C 180,E1 18422.514,E2 18422.514} C_VEL
LIN {X 0,Y 385.619,Z 607.707,A -85,B 0,C 180,E1 18418.415,E2 18418.415} C_VEL
LIN {X 0,Y 385.622,Z 607.762,A -85,B 0,C 180,E1 18414.31,E2 18414.31} C_VEL
LIN {X 0,Y 385.628,Z 607.765,A -85,B 0,C 180,E1 18410.176,E2 18410.176} C_VEL
LIN {X 0,Y 385.616,Z 607.745,A -85,B 0,C 180,E1 18406.123,E2 18406.123} C_VEL
LIN {X 0,Y 385.609,Z 607.747,A -85,B 0,C 180,E1 18402.133,E2 18402.133} C_VEL
LIN {X 0,Y 385.604,Z 607.762,A -85,B 0,C 180,E1 18398.107,E2 18398.107} C_VEL
LIN {X 0,Y 385.598,Z 607.737,A -85,B 0,C 180,E1 18394.062,E2 18394.062} C_VEL
LIN {X 0,Y 385.597,Z 607.764,A -85,B 0,C 180,E1 18389.994,E2 18389.994} C_VEL
LIN {X 0,Y 385.595,Z 607.73,A -85,B 0,C 180,E1 18385.991,E2 18385.991} C_VEL
LIN {X 0,Y 385.599,Z 607.763,A -85,B 0,C 180,E1 18381.925,E2 18381.925} C_VEL
LIN {X 0,Y 385.602,Z 607.729,A -85,B 0,C 180,E1 18377.973,E2 18377.973} C_VEL
LIN {X 0,Y 385.615,Z 607.76,A -85,B 0,C 180,E1 18373.954,E2 18373.954} C_VEL
LIN {X 0,Y 385.618,Z 607.734,A -85,B 0,C 180,E1 18370.005,E2 18370.005} C_VEL
LIN {X 0,Y 385.627,Z 607.758,A -85,B 0,C 180,E1 18365.953,E2 18365.953} C_VEL
LIN {X 0,Y 385.622,Z 607.737,A -85,B 0,C 180,E1 18361.932,E2 18361.932} C_VEL
LIN {X 0,Y 385.619,Z 607.756,A -85,B 0,C 180,E1 18357.92,E2 18357.92} C_VEL
LIN {X 0,Y 385.61,Z 607.74,A -85,B 0,C 180,E1 18353.898,E2 18353.898} C_VEL
LIN {X 0,Y 385.594,Z 607.761,A -85,B 0,C 180,E1 18349.995,E2 18349.995} C_VEL
LIN {X 0,Y 385.58,Z 607.745,A -85,B 0,C 180,E1 18346.045,E2 18346.045} C_VEL
LIN {X 0,Y 385.582,Z 607.768,A -85,B 0,C 180,E1 18342.027,E2 18342.027} C_VEL
LIN {X 0,Y 385.577,Z 607.757,A -85,B 0,C 180,E1 18338.074,E2 18338.074} C_VEL
LIN {X 0,Y 385.589,Z 607.747,A -85,B 0,C 180,E1 18334.132,E2 18334.132} C_VEL
LIN {X 0,Y 385.611,Z 607.757,A -85,B 0,C 180,E1 18330.301,E2 18330.301} C_VEL
LIN {X 0,Y 385.617,Z 607.759,A -85,B 0,C 180,E1 18326.298,E2 18326.298} C_VEL
LIN {X 0,Y 385.628,Z 607.756,A -85,B 0,C 180,E1 18322.262,E2 18322.262} C_VEL
LIN {X 0,Y 385.626,Z 607.754,A -85,B 0,C 180,E1 18318.214,E2 18318.214} C_VEL
LIN {X 0,Y 385.628,Z 607.976,A -85,B 0,C 180,E1 18314.413,E2 18314.413} C_VEL
LIN {X 0,Y 392.716,Z 627.101,A -85,B 0,C 180,E1 18311.095,E2 18311.095} C_VEL
LIN {X 0,Y 400.03,Z 648.255,A -85,B 0,C 180,E1 18307.831,E2 18307.831} C_VEL
LIN {X 0,Y 402.774,Z 657.062,A -85,B 0,C 180,E1 18306.569,E2 18306.569} C_VEL
LIN {X 0,Y 398.499,Z 694.533,A -85,B 0,C 180,E1 18302.708,E2 18302.708} C_VEL
LIN {X 0,Y 401.33,Z 721.731,A -85,B 0,C 180,E1 18301.985,E2 18301.985} C_VEL
LIN {X 0,Y 398.096,Z 891.145,A -85,B 0,C 180,E1 18298.951,E2 18298.951} C_VEL
LIN {X 0,Y 397.074,Z 909.785,A -85,B 0,C 180,E1 18298.368,E2 18298.368} C_VEL
LIN {X 0,Y 395.726,Z 927.742,A -85,B 0,C 180,E1 18297.541,E2 18297.541} C_VEL
LIN {X 0,Y 394.059,Z 945.971,A -85,B 0,C 180,E1 18296.405,E2 18296.405} C_VEL
LIN {X 0,Y 392.387,Z 962.217,A -85,B 0,C 180,E1 18295.105,E2 18295.105} C_VEL
LIN {X 0,Y 390.61,Z 978.041,A -85,B 0,C 180,E1 18293.536,E2 18293.536} C_VEL
LIN {X 0,Y 388.951,Z 992.934,A -85,B 0,C 180,E1 18291.727,E2 18291.727} C_VEL
LIN {X 0,Y 387.487,Z 1006.313,A -85,B 0,C 180,E1 18289.757,E2 18289.757} C_VEL
LIN {X 0,Y 386.216,Z 1019.067,A -85,B 0,C 180,E1 18287.476,E2 18287.476} C_VEL
LIN {X 0,Y 385.317,Z 1030.164,A -85,B 0,C 180,E1 18285.04,E2 18285.04} C_VEL
LIN {X 0,Y 384.802,Z 1039.151,A -85,B 0,C 180,E1 18282.607,E2 18282.607} C_VEL
LIN {X 0,Y 384.599,Z 1046.674,A -85,B 0,C 180,E1 18280.031,E2 18280.031} C_VEL
LIN {X 0,Y 384.638,Z 1052.347,A -85,B 0,C 180,E1 18277.468,E2 18277.468} C_VEL
LIN {X 0,Y 384.779,Z 1056.303,A -85,B 0,C 180,E1 18274.92,E2 18274.92} C_VEL
LIN {X 0,Y 384.927,Z 1058.621,A -85,B 0,C 180,E1 18272.382,E2 18272.382} C_VEL
LIN {X 0,Y 384.988,Z 1059.344,A -85,B 0,C 180,E1 18269.851,E2 18269.851} C_VEL
LIN {X 0,Y 384.909,Z 1058.45,A -85,B 0,C 180,E1 18267.32,E2 18267.32} C_VEL
LIN {X 0,Y 384.757,Z 1055.958,A -85,B 0,C 180,E1 18264.782,E2 18264.782} C_VEL
LIN {X 0,Y 384.616,Z 1051.844,A -85,B 0,C 180,E1 18262.231,E2 18262.231} C_VEL
LIN {X 0,Y 384.596,Z 1046.034,A -85,B 0,C 180,E1 18259.666,E2 18259.666} C_VEL
LIN {X 0,Y 384.833,Z 1038.414,A -85,B 0,C 180,E1 18257.089,E2 18257.089} C_VEL
LIN {X 0,Y 385.393,Z 1029.389,A -85,B 0,C 180,E1 18254.655,E2 18254.655} C_VEL
LIN {X 0,Y 386.361,Z 1018.309,A -85,B 0,C 180,E1 18252.22,E2 18252.22} C_VEL
LIN {X 0,Y 387.719,Z 1005.652,A -85,B 0,C 180,E1 18249.941,E2 18249.941} C_VEL
LIN {X 0,Y 389.339,Z 991.853,A -85,B 0,C 180,E1 18247.9,E2 18247.9} C_VEL
LIN {X 0,Y 391.12,Z 977.087,A -85,B 0,C 180,E1 18246.097,E2 18246.097} C_VEL
LIN {X 0,Y 393.032,Z 961.501,A -85,B 0,C 180,E1 18244.537,E2 18244.537} C_VEL
LIN {X 0,Y 394.949,Z 944.344,A -85,B 0,C 180,E1 18243.157,E2 18243.157} C_VEL
LIN {X 0,Y 396.723,Z 926.531,A -85,B 0,C 180,E1 18242.045,E2 18242.045} C_VEL
LIN {X 0,Y 398.228,Z 908.38,A -85,B 0,C 180,E1 18241.21,E2 18241.21} C_VEL
LIN {X 0,Y 399.32,Z 889.724,A -85,B 0,C 180,E1 18240.63,E2 18240.63} C_VEL
LIN {X 0,Y 402.831,Z 719.112,A -85,B 0,C 180,E1 18237.497,E2 18237.497} C_VEL
LIN {X 0,Y 400.115,Z 694.402,A -85,B 0,C 180,E1 18236.72,E2 18236.72} C_VEL
LIN {X 0,Y 404.832,Z 659.132,A -85,B 0,C 180,E1 18232.916,E2 18232.916} C_VEL
LIN {X 0,Y 399.723,Z 643.124,A -85,B 0,C 180,E1 18230.28,E2 18230.28} C_VEL
LIN {X 0,Y 394.296,Z 628.661,A -85,B 0,C 180,E1 18227.554,E2 18227.554} C_VEL
LIN {X 0,Y 388.921,Z 615.656,A -85,B 0,C 180,E1 18224.782,E2 18224.782} C_VEL
LIN {X 0,Y 385.601,Z 607.981,A -85,B 0,C 180,E1 18222.91,E2 18222.91} C_VEL
LIN {X 0,Y 385.598,Z 607.76,A -85,B 0,C 180,E1 18219.402,E2 18219.402} C_VEL
LIN {X 0,Y 385.614,Z 607.751,A -85,B 0,C 180,E1 18215.495,E2 18215.495} C_VEL
LIN {X 0,Y 385.627,Z 607.747,A -85,B 0,C 180,E1 18211.41,E2 18211.41} C_VEL
LIN {X 0,Y 385.62,Z 607.746,A -85,B 0,C 180,E1 18207.486,E2 18207.486} C_VEL
LIN {X 0,Y 385.603,Z 607.746,A -85,B 0,C 180,E1 18203.535,E2 18203.535} C_VEL
LIN {X 0,Y 385.585,Z 607.751,A -85,B 0,C 180,E1 18199.7,E2 18199.7} C_VEL
LIN {X 0,Y 385.58,Z 607.763,A -85,B 0,C 180,E1 18195.8,E2 18195.8} C_VEL
LIN {X 0,Y 385.581,Z 607.768,A -85,B 0,C 180,E1 18191.821,E2 18191.821} C_VEL
LIN {X 0,Y 385.589,Z 607.76,A -85,B 0,C 180,E1 18187.882,E2 18187.882} C_VEL
LIN {X 0,Y 385.601,Z 607.746,A -85,B 0,C 180,E1 18184.014,E2 18184.014} C_VEL
LIN {X 0,Y 385.619,Z 607.743,A -85,B 0,C 180,E1 18180,E2 18180} C_VEL
LIN {X 0,Y 385.619,Z 607.748,A -85,B 0,C 180,E1 18175.985,E2 18175.985} C_VEL
LIN {X 0,Y 385.629,Z 607.753,A -85,B 0,C 180,E1 18171.951,E2 18171.951} C_VEL
LIN {X 0,Y 385.624,Z 607.757,A -85,B 0,C 180,E1 18167.822,E2 18167.822} C_VEL
LIN {X 0,Y 385.618,Z 607.759,A -85,B 0,C 180,E1 18163.892,E2 18163.892} C_VEL
LIN {X 0,Y 385.614,Z 607.754,A -85,B 0,C 180,E1 18159.823,E2 18159.823} C_VEL
LIN {X 0,Y 385.603,Z 607.753,A -85,B 0,C 180,E1 18155.885,E2 18155.885} C_VEL
LIN {X 0,Y 385.637,Z 608.014,A -85,B 0,C 180,E1 18152.371,E2 18152.371} C_VEL
LIN {X 0,Y 390.291,Z 620.471,A -85,B 0,C 180,E1 18149.007,E2 18149.007} C_VEL
LIN {X 0,Y 394.534,Z 633.148,A -85,B 0,C 180,E1 18145.938,E2 18145.938} C_VEL
LIN {X 0,Y 398.371,Z 646.756,A -85,B 0,C 180,E1 18142.953,E2 18142.953} C_VEL
LIN {X 0,Y 399.824,Z 653.932,A -85,B 0,C 180,E1 18141.512,E2 18141.512} C_VEL
LIN {X 0,Y 396.348,Z 681.075,A -85,B 0,C 180,E1 18137.231,E2 18137.231} C_VEL
LIN {X 0,Y 393.525,Z 706.86,A -85,B 0,C 180,E1 18133.244,E2 18133.244} C_VEL
LIN {X 0,Y 395.911,Z 718.822,A -85,B 0,C 180,E1 18132.726,E2 18132.726} C_VEL
LIN {X 0,Y 399.086,Z 737.283,A -85,B 0,C 180,E1 18132.065,E2 18132.065} C_VEL
LIN {X 0,Y 396.685,Z 832.698,A -85,B 0,C 180,E1 18130.155,E2 18130.155} C_VEL
LIN {X 0,Y 396.023,Z 848.928,A -85,B 0,C 180,E1 18129.55,E2 18129.55} C_VEL
LIN {X 0,Y 395.094,Z 863.345,A -85,B 0,C 180,E1 18128.748,E2 18128.748} C_VEL
LIN {X 0,Y 393.814,Z 878.234,A -85,B 0,C 180,E1 18127.613,E2 18127.613} C_VEL
LIN {X 0,Y 392.359,Z 891.75,A -85,B 0,C 180,E1 18126.243,E2 18126.243} C_VEL
LIN {X 0,Y 390.976,Z 903.143,A -85,B 0,C 180,E1 18124.77,E2 18124.77} C_VEL
LIN {X 0,Y 389.486,Z 914.365,A -85,B 0,C 180,E1 18122.917,E2 18122.917} C_VEL
LIN {X 0,Y 388.163,Z 923.618,A -85,B 0,C 180,E1 18120.933,E2 18120.933} C_VEL
LIN {X 0,Y 387.113,Z 930.942,A -85,B 0,C 180,E1 18118.881,E2 18118.881} C_VEL
LIN {X 0,Y 386.285,Z 936.837,A -85,B 0,C 180,E1 18116.602,E2 18116.602} C_VEL
LIN {X 0,Y 385.758,Z 940.709,A -85,B 0,C 180,E1 18114.338,E2 18114.338} C_VEL
LIN {X 0,Y 385.457,Z 942.913,A -85,B 0,C 180,E1 18111.933,E2 18111.933} C_VEL
LIN {X 0,Y 385.349,Z 943.183,A -85,B 0,C 180,E1 18109.555,E2 18109.555} C_VEL
LIN {X 0,Y 385.412,Z 941.808,A -85,B 0,C 180,E1 18107.312,E2 18107.312} C_VEL
LIN {X 0,Y 385.68,Z 938.361,A -85,B 0,C 180,E1 18104.871,E2 18104.871} C_VEL
LIN {X 0,Y 386.138,Z 933.487,A -85,B 0,C 180,E1 18102.715,E2 18102.715} C_VEL
LIN {X 0,Y 386.855,Z 926.771,A -85,B 0,C 180,E1 18100.574,E2 18100.574} C_VEL
LIN {X 0,Y 387.781,Z 918.49,A -85,B 0,C 180,E1 18098.6,E2 18098.6} C_VEL
LIN {X 0,Y 388.882,Z 908.803,A -85,B 0,C 180,E1 18096.792,E2 18096.792} C_VEL
LIN {X 0,Y 389.721,Z 900.948,A -85,B 0,C 180,E1 18095.597,E2 18095.597} C_VEL
LIN {X 0,Y 389.369,Z 895.405,A -85,B 0,C 180,E1 18094.798,E2 18094.798} C_VEL
LIN {X 0,Y 386.187,Z 884.946,A -85,B 0,C 180,E1 18093.381,E2 18093.381} C_VEL
LIN {X 0,Y 384.754,Z 877.951,A -85,B 0,C 180,E1 18092.599,E2 18092.599} C_VEL
LIN {X 0,Y 384.743,Z 874.128,A -85,B 0,C 180,E1 18092.254,E2 18092.254} C_VEL
LIN {X 0,Y 385.76,Z 860.363,A -85,B 0,C 180,E1 18091.262,E2 18091.262} C_VEL
LIN {X 0,Y 386.624,Z 843.998,A -85,B 0,C 180,E1 18090.421,E2 18090.421} C_VEL
LIN {X 0,Y 387.1,Z 827.943,A -85,B 0,C 180,E1 18089.907,E2 18089.907} C_VEL
LIN {X 0,Y 388.9,Z 735.032,A -85,B 0,C 180,E1 18088.084,E2 18088.084} C_VEL
LIN {X 0,Y 384.099,Z 707.114,A -85,B 0,C 180,E1 18087.165,E2 18087.165} C_VEL
LIN {X 0,Y 386.775,Z 678.898,A -85,B 0,C 180,E1 18082.872,E2 18082.872} C_VEL
LIN {X 0,Y 389.811,Z 651.37,A -85,B 0,C 180,E1 18078.609,E2 18078.609} C_VEL
LIN {X 0,Y 386.1,Z 636.576,A -85,B 0,C 180,E1 18075.758,E2 18075.758} C_VEL
LIN {X 0,Y 381.328,Z 620.395,A -85,B 0,C 180,E1 18072.45,E2 18072.45} C_VEL
LIN {X 0,Y 377.689,Z 608.859,A -85,B 0,C 180,E1 18069.87,E2 18069.87} C_VEL
LIN {X 0,Y 377.67,Z 608.705,A -85,B 0,C 180,E1 18065.772,E2 18065.772} C_VEL
LIN {X 0,Y 377.68,Z 608.737,A -85,B 0,C 180,E1 18061.713,E2 18061.713} C_VEL
LIN {X 0,Y 377.674,Z 608.706,A -85,B 0,C 180,E1 18057.622,E2 18057.622} C_VEL
LIN {X 0,Y 377.681,Z 608.746,A -85,B 0,C 180,E1 18053.591,E2 18053.591} C_VEL
LIN {X 0,Y 377.692,Z 608.75,A -85,B 0,C 180,E1 18049.445,E2 18049.445} C_VEL
LIN {X 0,Y 377.681,Z 608.748,A -85,B 0,C 180,E1 18045.234,E2 18045.234} C_VEL
LIN {X 0,Y 377.69,Z 608.722,A -85,B 0,C 180,E1 18041.238,E2 18041.238} C_VEL
LIN {X 0,Y 377.686,Z 608.75,A -85,B 0,C 180,E1 18037.128,E2 18037.128} C_VEL
LIN {X 0,Y 377.686,Z 608.724,A -85,B 0,C 180,E1 18033.049,E2 18033.049} C_VEL
LIN {X 0,Y 377.692,Z 608.745,A -85,B 0,C 180,E1 18028.977,E2 18028.977} C_VEL
LIN {X 0,Y 377.683,Z 608.722,A -85,B 0,C 180,E1 18024.894,E2 18024.894} C_VEL
LIN {X 0,Y 377.689,Z 608.746,A -85,B 0,C 180,E1 18020.778,E2 18020.778} C_VEL
LIN {X 0,Y 377.681,Z 608.719,A -85,B 0,C 180,E1 18016.614,E2 18016.614} C_VEL
LIN {X 0,Y 377.675,Z 608.752,A -85,B 0,C 180,E1 18012.694,E2 18012.694} C_VEL
LIN {X 0,Y 377.661,Z 608.716,A -85,B 0,C 180,E1 18008.68,E2 18008.68} C_VEL
LIN {X 0,Y 377.654,Z 608.753,A -85,B 0,C 180,E1 18004.708,E2 18004.708} C_VEL
LIN {X 0,Y 377.642,Z 608.72,A -85,B 0,C 180,E1 18000.759,E2 18000.759} C_VEL
LIN {X 0,Y 377.647,Z 608.754,A -85,B 0,C 180,E1 17996.661,E2 17996.661} C_VEL
LIN {X 0,Y 377.64,Z 608.723,A -85,B 0,C 180,E1 17992.546,E2 17992.546} C_VEL
LIN {X 0,Y 377.648,Z 608.754,A -85,B 0,C 180,E1 17988.547,E2 17988.547} C_VEL
LIN {X 0,Y 377.651,Z 608.738,A -85,B 0,C 180,E1 17984.521,E2 17984.521} C_VEL
LIN {X 0,Y 377.66,Z 608.743,A -85,B 0,C 180,E1 17980.514,E2 17980.514} C_VEL
LIN {X 0,Y 377.677,Z 608.752,A -85,B 0,C 180,E1 17976.603,E2 17976.603} C_VEL
LIN {X 0,Y 377.682,Z 608.744,A -85,B 0,C 180,E1 17972.483,E2 17972.483} C_VEL
LIN {X 0,Y 377.686,Z 608.738,A -85,B 0,C 180,E1 17968.479,E2 17968.479} C_VEL
LIN {X 0,Y 377.681,Z 608.742,A -85,B 0,C 180,E1 17964.365,E2 17964.365} C_VEL
LIN {X 0,Y 377.691,Z 608.747,A -85,B 0,C 180,E1 17960.358,E2 17960.358} C_VEL
LIN {X 0,Y 377.677,Z 608.748,A -85,B 0,C 180,E1 17956.282,E2 17956.282} C_VEL
LIN {X 0,Y 377.695,Z 609.131,A -85,B 0,C 180,E1 17955.165,E2 17955.165} C_VEL
LIN {X 0,Y 384.798,Z 628.169,A -85,B 0,C 180,E1 17951.778,E2 17951.778} C_VEL
LIN {X 0,Y 391.633,Z 647.839,A -85,B 0,C 180,E1 17948.627,E2 17948.627} C_VEL
LIN {X 0,Y 395.376,Z 659.689,A -85,B 0,C 180,E1 17946.884,E2 17946.884} C_VEL
LIN {X 0,Y 391.173,Z 694.308,A -85,B 0,C 180,E1 17943.227,E2 17943.227} C_VEL
LIN {X 0,Y 394.025,Z 722.636,A -85,B 0,C 180,E1 17942.446,E2 17942.446} C_VEL
LIN {X 0,Y 390.657,Z 890.663,A -85,B 0,C 180,E1 17939.386,E2 17939.386} C_VEL
LIN {X 0,Y 389.612,Z 909.229,A -85,B 0,C 180,E1 17938.794,E2 17938.794} C_VEL
LIN {X 0,Y 388.175,Z 927.557,A -85,B 0,C 180,E1 17937.933,E2 17937.933} C_VEL
LIN {X 0,Y 386.49,Z 945.259,A -85,B 0,C 180,E1 17936.808,E2 17936.808} C_VEL
LIN {X 0,Y 384.74,Z 961.637,A -85,B 0,C 180,E1 17935.474,E2 17935.474} C_VEL
LIN {X 0,Y 382.886,Z 977.398,A -85,B 0,C 180,E1 17933.877,E2 17933.877} C_VEL
LIN {X 0,Y 381.15,Z 992.234,A -85,B 0,C 180,E1 17932.033,E2 17932.033} C_VEL
LIN {X 0,Y 379.624,Z 1005.56,A -85,B 0,C 180,E1 17930.023,E2 17930.023} C_VEL
LIN {X 0,Y 378.3,Z 1018.243,A -85,B 0,C 180,E1 17927.695,E2 17927.695} C_VEL
LIN {X 0,Y 377.403,Z 1028.751,A -85,B 0,C 180,E1 17925.346,E2 17925.346} C_VEL
LIN {X 0,Y 376.858,Z 1037.742,A -85,B 0,C 180,E1 17922.878,E2 17922.878} C_VEL
LIN {X 0,Y 376.639,Z 1045.335,A -85,B 0,C 180,E1 17920.246,E2 17920.246} C_VEL
LIN {X 0,Y 376.683,Z 1051.068,A -85,B 0,C 180,E1 17917.627,E2 17917.627} C_VEL
LIN {X 0,Y 376.847,Z 1055.066,A -85,B 0,C 180,E1 17915.023,E2 17915.023} C_VEL
LIN {X 0,Y 377.009,Z 1057.413,A -85,B 0,C 180,E1 17912.432,E2 17912.432} C_VEL
LIN {X 0,Y 377.078,Z 1058.15,A -85,B 0,C 180,E1 17909.848,E2 17909.848} C_VEL
LIN {X 0,Y 376.988,Z 1057.259,A -85,B 0,C 180,E1 17907.264,E2 17907.264} C_VEL
LIN {X 0,Y 376.813,Z 1054.77,A -85,B 0,C 180,E1 17904.671,E2 17904.671} C_VEL
LIN {X 0,Y 376.648,Z 1050.466,A -85,B 0,C 180,E1 17901.961,E2 17901.961} C_VEL
LIN {X 0,Y 376.631,Z 1044.461,A -85,B 0,C 180,E1 17899.291,E2 17899.291} C_VEL
LIN {X 0,Y 376.912,Z 1036.72,A -85,B 0,C 180,E1 17896.657,E2 17896.657} C_VEL
LIN {X 0,Y 377.587,Z 1026.931,A -85,B 0,C 180,E1 17894.015,E2 17894.015} C_VEL
LIN {X 0,Y 378.702,Z 1015.496,A -85,B 0,C 180,E1 17891.529,E2 17891.529} C_VEL
LIN {X 0,Y 380.102,Z 1003.41,A -85,B 0,C 180,E1 17889.361,E2 17889.361} C_VEL
LIN {X 0,Y 381.865,Z 989.444,A -85,B 0,C 180,E1 17887.283,E2 17887.283} C_VEL
LIN {X 0,Y 383.798,Z 974.453,A -85,B 0,C 180,E1 17885.448,E2 17885.448} C_VEL
LIN {X 0,Y 385.853,Z 958.526,A -85,B 0,C 180,E1 17883.863,E2 17883.863} C_VEL
LIN {X 0,Y 387.828,Z 941.637,A -85,B 0,C 180,E1 17882.518,E2 17882.518} C_VEL
LIN {X 0,Y 389.547,Z 924.984,A -85,B 0,C 180,E1 17881.484,E2 17881.484} C_VEL
LIN {X 0,Y 391.124,Z 906.885,A -85,B 0,C 180,E1 17880.652,E2 17880.652} C_VEL
LIN {X 0,Y 392.24,Z 887.957,A -85,B 0,C 180,E1 17880.066,E2 17880.066} C_VEL
LIN {X 0,Y 395.881,Z 719.997,A -85,B 0,C 180,E1 17876.934,E2 17876.934} C_VEL
LIN {X 0,Y 393.137,Z 694.579,A -85,B 0,C 180,E1 17876.109,E2 17876.109} C_VEL
LIN {X 0,Y 397.749,Z 662.081,A -85,B 0,C 180,E1 17872.531,E2 17872.531} C_VEL
LIN {X 0,Y 392.881,Z 646.656,A -85,B 0,C 180,E1 17869.919,E2 17869.919} C_VEL
LIN {X 0,Y 387.4,Z 631.886,A -85,B 0,C 180,E1 17867.049,E2 17867.049} C_VEL
LIN {X 0,Y 382.502,Z 620.178,A -85,B 0,C 180,E1 17864.47,E2 17864.47} C_VEL
LIN {X 0,Y 378.891,Z 612.151,A -85,B 0,C 180,E1 17862.497,E2 17862.497} C_VEL
LIN {X 0,Y 377.69,Z 608.906,A -85,B 0,C 180,E1 17861.608,E2 17861.608} C_VEL
LIN {X 0,Y 377.684,Z 608.743,A -85,B 0,C 180,E1 17857.669,E2 17857.669} C_VEL
LIN {X 0,Y 377.685,Z 608.754,A -85,B 0,C 180,E1 17853.497,E2 17853.497} C_VEL
LIN {X 0,Y 377.695,Z 608.751,A -85,B 0,C 180,E1 17849.431,E2 17849.431} C_VEL
LIN {X 0,Y 377.683,Z 608.751,A -85,B 0,C 180,E1 17845.228,E2 17845.228} C_VEL
LIN {X 0,Y 377.691,Z 608.753,A -85,B 0,C 180,E1 17841.102,E2 17841.102} C_VEL
LIN {X 0,Y 377.685,Z 608.75,A -85,B 0,C 180,E1 17836.93,E2 17836.93} C_VEL
LIN {X 0,Y 377.683,Z 608.744,A -85,B 0,C 180,E1 17832.848,E2 17832.848} C_VEL
LIN {X 0,Y 377.683,Z 608.731,A -85,B 0,C 180,E1 17828.679,E2 17828.679} C_VEL
LIN {X 0,Y 377.671,Z 608.731,A -85,B 0,C 180,E1 17824.707,E2 17824.707} C_VEL
LIN {X 0,Y 377.671,Z 608.737,A -85,B 0,C 180,E1 17820.606,E2 17820.606} C_VEL
LIN {X 0,Y 377.664,Z 608.748,A -85,B 0,C 180,E1 17816.583,E2 17816.583} C_VEL
LIN {X 0,Y 377.661,Z 608.754,A -85,B 0,C 180,E1 17812.546,E2 17812.546} C_VEL
LIN {X 0,Y 377.656,Z 608.756,A -85,B 0,C 180,E1 17808.547,E2 17808.547} C_VEL
LIN {X 0,Y 377.653,Z 608.756,A -85,B 0,C 180,E1 17804.49,E2 17804.49} C_VEL
LIN {X 0,Y 377.657,Z 608.752,A -85,B 0,C 180,E1 17800.352,E2 17800.352} C_VEL
LIN {X 0,Y 377.655,Z 608.743,A -85,B 0,C 180,E1 17796.27,E2 17796.27} C_VEL
LIN {X 0,Y 377.716,Z 609.036,A -85,B 0,C 180,E1 17793.584,E2 17793.584} C_VEL
LIN {X 0,Y 381.8,Z 619.77,A -85,B 0,C 180,E1 17790.505,E2 17790.505} C_VEL
LIN {X 0,Y 386.218,Z 632.456,A -85,B 0,C 180,E1 17787.243,E2 17787.243} C_VEL
LIN {X 0,Y 390.074,Z 645.393,A -85,B 0,C 180,E1 17784.237,E2 17784.237} C_VEL
LIN {X 0,Y 392.68,Z 656.474,A -85,B 0,C 180,E1 17781.886,E2 17781.886} C_VEL
LIN {X 0,Y 389.014,Z 683.649,A -85,B 0,C 180,E1 17777.532,E2 17777.532} C_VEL
LIN {X 0,Y 386.365,Z 706.741,A -85,B 0,C 180,E1 17773.911,E2 17773.911} C_VEL
LIN {X 0,Y 389.089,Z 720.403,A -85,B 0,C 180,E1 17773.304,E2 17773.304} C_VEL
LIN {X 0,Y 392.176,Z 738.476,A -85,B 0,C 180,E1 17772.636,E2 17772.636} C_VEL
LIN {X 0,Y 389.637,Z 833.222,A -85,B 0,C 180,E1 17770.701,E2 17770.701} C_VEL
LIN {X 0,Y 388.941,Z 849.32,A -85,B 0,C 180,E1 17770.094,E2 17770.094} C_VEL
LIN {X 0,Y 388.035,Z 862.983,A -85,B 0,C 180,E1 17769.336,E2 17769.336} C_VEL
LIN {X 0,Y 386.746,Z 877.26,A -85,B 0,C 180,E1 17768.256,E2 17768.256} C_VEL
LIN {X 0,Y 385.357,Z 889.979,A -85,B 0,C 180,E1 17767.01,E2 17767.01} C_VEL
LIN {X 0,Y 383.753,Z 902.558,A -85,B 0,C 180,E1 17765.422,E2 17765.422} C_VEL
LIN {X 0,Y 382.287,Z 913.108,A -85,B 0,C 180,E1 17763.723,E2 17763.723} C_VEL
LIN {X 0,Y 380.816,Z 922.904,A -85,B 0,C 180,E1 17761.713,E2 17761.713} C_VEL
LIN {X 0,Y 379.609,Z 930.602,A -85,B 0,C 180,E1 17759.634,E2 17759.634} C_VEL
LIN {X 0,Y 378.705,Z 936.566,A -85,B 0,C 180,E1 17757.487,E2 17757.487} C_VEL
LIN {X 0,Y 378.007,Z 941.182,A -85,B 0,C 180,E1 17755.037,E2 17755.037} C_VEL
LIN {X 0,Y 377.632,Z 943.67,A -85,B 0,C 180,E1 17752.741,E2 17752.741} C_VEL
LIN {X 0,Y 377.455,Z 944.503,A -85,B 0,C 180,E1 17750.304,E2 17750.304} C_VEL
LIN {X 0,Y 377.464,Z 943.501,A -85,B 0,C 180,E1 17747.895,E2 17747.895} C_VEL
LIN {X 0,Y 377.677,Z 940.72,A -85,B 0,C 180,E1 17745.494,E2 17745.494} C_VEL
LIN {X 0,Y 378.12,Z 936.05,A -85,B 0,C 180,E1 17743.144,E2 17743.144} C_VEL
LIN {X 0,Y 378.8,Z 929.812,A -85,B 0,C 180,E1 17740.955,E2 17740.955} C_VEL
LIN {X 0,Y 379.788,Z 921.481,A -85,B 0,C 180,E1 17738.783,E2 17738.783} C_VEL
LIN {X 0,Y 380.983,Z 911.375,A -85,B 0,C 180,E1 17736.782,E2 17736.782} C_VEL
LIN {X 0,Y 382.193,Z 900.57,A -85,B 0,C 180,E1 17735.103,E2 17735.103} C_VEL
LIN {X 0,Y 383.461,Z 888.231,A -85,B 0,C 180,E1 17733.588,E2 17733.588} C_VEL
LIN {X 0,Y 384.692,Z 874.75,A -85,B 0,C 180,E1 17732.306,E2 17732.306} C_VEL
LIN {X 0,Y 384.743,Z 874.128,A -85,B 0,C 180,E1 17732.254,E2 17732.254} C_VEL
LIN {X 0,Y 384.35,Z 867.411,A -85,B 0,C 180,E1 17731.672,E2 17731.672} C_VEL
LIN {X 0,Y 380.781,Z 854.112,A -85,B 0,C 180,E1 17730.553,E2 17730.553} C_VEL
LIN {X 0,Y 379.34,Z 846.01,A -85,B 0,C 180,E1 17730.05,E2 17730.05} C_VEL
LIN {X 0,Y 379.283,Z 842.821,A -85,B 0,C 180,E1 17729.91,E2 17729.91} C_VEL
LIN {X 0,Y 379.764,Z 826.107,A -85,B 0,C 180,E1 17729.399,E2 17729.399} C_VEL
LIN {X 0,Y 381.614,Z 736.195,A -85,B 0,C 180,E1 17727.611,E2 17727.611} C_VEL
LIN {X 0,Y 376.657,Z 707.367,A -85,B 0,C 180,E1 17726.652,E2 17726.652} C_VEL
LIN {X 0,Y 376.848,Z 703.966,A -85,B 0,C 180,E1 17726.196,E2 17726.196} C_VEL
LIN {X 0,Y 379.765,Z 675.944,A -85,B 0,C 180,E1 17721.826,E2 17721.826} C_VEL
LIN {X 0,Y 382.315,Z 653.171,A -85,B 0,C 180,E1 17718.229,E2 17718.229} C_VEL
LIN {X 0,Y 377.764,Z 635.909,A -85,B 0,C 180,E1 17714.809,E2 17714.809} C_VEL
LIN {X 0,Y 372.935,Z 619.82,A -85,B 0,C 180,E1 17711.394,E2 17711.394} C_VEL
LIN {X 0,Y 369.762,Z 609.861,A -85,B 0,C 180,E1 17709.087,E2 17709.087} C_VEL
LIN {X 0,Y 369.736,Z 609.7,A -85,B 0,C 180,E1 17704.949,E2 17704.949} C_VEL
LIN {X 0,Y 369.74,Z 609.699,A -85,B 0,C 180,E1 17700.865,E2 17700.865} C_VEL
LIN {X 0,Y 369.736,Z 609.718,A -85,B 0,C 180,E1 17696.681,E2 17696.681} C_VEL
LIN {X 0,Y 369.735,Z 609.725,A -85,B 0,C 180,E1 17692.521,E2 17692.521} C_VEL
LIN {X 0,Y 369.729,Z 609.733,A -85,B 0,C 180,E1 17688.504,E2 17688.504} C_VEL
LIN {X 0,Y 369.731,Z 609.741,A -85,B 0,C 180,E1 17684.443,E2 17684.443} C_VEL
LIN {X 0,Y 369.724,Z 609.714,A -85,B 0,C 180,E1 17680.267,E2 17680.267} C_VEL
LIN {X 0,Y 369.724,Z 609.737,A -85,B 0,C 180,E1 17676.125,E2 17676.125} C_VEL
LIN {X 0,Y 369.721,Z 609.728,A -85,B 0,C 180,E1 17672.01,E2 17672.01} C_VEL
LIN {X 0,Y 369.72,Z 609.728,A -85,B 0,C 180,E1 17667.896,E2 17667.896} C_VEL
LIN {X 0,Y 369.716,Z 609.73,A -85,B 0,C 180,E1 17663.763,E2 17663.763} C_VEL
LIN {X 0,Y 369.716,Z 609.727,A -85,B 0,C 180,E1 17659.594,E2 17659.594} C_VEL
LIN {X 0,Y 369.714,Z 609.727,A -85,B 0,C 180,E1 17655.53,E2 17655.53} C_VEL
LIN {X 0,Y 369.719,Z 609.736,A -85,B 0,C 180,E1 17651.545,E2 17651.545} C_VEL
LIN {X 0,Y 369.72,Z 609.718,A -85,B 0,C 180,E1 17647.459,E2 17647.459} C_VEL
LIN {X 0,Y 369.724,Z 609.735,A -85,B 0,C 180,E1 17643.411,E2 17643.411} C_VEL
LIN {X 0,Y 369.73,Z 609.715,A -85,B 0,C 180,E1 17639.381,E2 17639.381} C_VEL
LIN {X 0,Y 369.738,Z 609.735,A -85,B 0,C 180,E1 17635.347,E2 17635.347} C_VEL
LIN {X 0,Y 369.742,Z 609.719,A -85,B 0,C 180,E1 17631.29,E2 17631.29} C_VEL
LIN {X 0,Y 369.746,Z 609.727,A -85,B 0,C 180,E1 17627.189,E2 17627.189} C_VEL
LIN {X 0,Y 369.747,Z 609.738,A -85,B 0,C 180,E1 17623.181,E2 17623.181} C_VEL
LIN {X 0,Y 369.746,Z 609.718,A -85,B 0,C 180,E1 17619.087,E2 17619.087} C_VEL
LIN {X 0,Y 369.734,Z 609.729,A -85,B 0,C 180,E1 17615.048,E2 17615.048} C_VEL
LIN {X 0,Y 369.73,Z 609.744,A -85,B 0,C 180,E1 17611.049,E2 17611.049} C_VEL
LIN {X 0,Y 369.713,Z 609.745,A -85,B 0,C 180,E1 17607.072,E2 17607.072} C_VEL
LIN {X 0,Y 369.702,Z 609.749,A -85,B 0,C 180,E1 17603.102,E2 17603.102} C_VEL
LIN {X 0,Y 369.696,Z 609.743,A -85,B 0,C 180,E1 17599.119,E2 17599.119} C_VEL
LIN {X 0,Y 369.783,Z 610.006,A -85,B 0,C 180,E1 17596.041,E2 17596.041} C_VEL
LIN {X 0,Y 376.725,Z 628.568,A -85,B 0,C 180,E1 17592.594,E2 17592.594} C_VEL
LIN {X 0,Y 383.657,Z 648.539,A -85,B 0,C 180,E1 17589.284,E2 17589.284} C_VEL
LIN {X 0,Y 387.984,Z 662.139,A -85,B 0,C 180,E1 17587.221,E2 17587.221} C_VEL
LIN {X 0,Y 383.878,Z 694.479,A -85,B 0,C 180,E1 17583.741,E2 17583.741} C_VEL
LIN {X 0,Y 386.746,Z 723.528,A -85,B 0,C 180,E1 17582.924,E2 17582.924} C_VEL
LIN {X 0,Y 383.244,Z 889.973,A -85,B 0,C 180,E1 17579.84,E2 17579.84} C_VEL
LIN {X 0,Y 382.168,Z 908.551,A -85,B 0,C 180,E1 17579.238,E2 17579.238} C_VEL
LIN {X 0,Y 380.694,Z 926.607,A -85,B 0,C 180,E1 17578.376,E2 17578.376} C_VEL
LIN {X 0,Y 378.933,Z 944.425,A -85,B 0,C 180,E1 17577.226,E2 17577.226} C_VEL
LIN {X 0,Y 377.101,Z 960.882,A -85,B 0,C 180,E1 17575.86,E2 17575.86} C_VEL
LIN {X 0,Y 375.169,Z 976.657,A -85,B 0,C 180,E1 17574.232,E2 17574.232} C_VEL
LIN {X 0,Y 373.294,Z 992.067,A -85,B 0,C 180,E1 17572.272,E2 17572.272} C_VEL
LIN {X 0,Y 371.657,Z 1005.759,A -85,B 0,C 180,E1 17570.132,E2 17570.132} C_VEL
LIN {X 0,Y 370.39,Z 1017.419,A -85,B 0,C 180,E1 17567.924,E2 17567.924} C_VEL
LIN {X 0,Y 369.459,Z 1027.811,A -85,B 0,C 180,E1 17565.541,E2 17565.541} C_VEL
LIN {X 0,Y 368.895,Z 1036.823,A -85,B 0,C 180,E1 17563.001,E2 17563.001} C_VEL
LIN {X 0,Y 368.679,Z 1044.368,A -85,B 0,C 180,E1 17560.311,E2 17560.311} C_VEL
LIN {X 0,Y 368.739,Z 1050.048,A -85,B 0,C 180,E1 17557.636,E2 17557.636} C_VEL
LIN {X 0,Y 368.926,Z 1053.989,A -85,B 0,C 180,E1 17554.976,E2 17554.976} C_VEL
LIN {X 0,Y 369.104,Z 1056.271,A -85,B 0,C 180,E1 17552.329,E2 17552.329} C_VEL
LIN {X 0,Y 369.163,Z 1056.935,A -85,B 0,C 180,E1 17549.69,E2 17549.69} C_VEL
LIN {X 0,Y 369.053,Z 1055.984,A -85,B 0,C 180,E1 17547.05,E2 17547.05} C_VEL
LIN {X 0,Y 368.84,Z 1053.216,A -85,B 0,C 180,E1 17544.244,E2 17544.244} C_VEL
LIN {X 0,Y 368.663,Z 1048.601,A -85,B 0,C 180,E1 17541.422,E2 17541.422} C_VEL
LIN {X 0,Y 368.674,Z 1042.471,A -85,B 0,C 180,E1 17538.74,E2 17538.74} C_VEL
LIN {X 0,Y 369.034,Z 1034.471,A -85,B 0,C 180,E1 17536.047,E2 17536.047} C_VEL
LIN {X 0,Y 369.761,Z 1025.04,A -85,B 0,C 180,E1 17533.505,E2 17533.505} C_VEL
LIN {X 0,Y 370.909,Z 1014.25,A -85,B 0,C 180,E1 17531.118,E2 17531.118} C_VEL
LIN {X 0,Y 372.403,Z 1002.223,A -85,B 0,C 180,E1 17528.914,E2 17528.914} C_VEL
LIN {X 0,Y 374.21,Z 988.8,A -85,B 0,C 180,E1 17526.873,E2 17526.873} C_VEL
LIN {X 0,Y 376.303,Z 973.535,A -85,B 0,C 180,E1 17524.966,E2 17524.966} C_VEL
LIN {X 0,Y 378.516,Z 957.218,A -85,B 0,C 180,E1 17523.317,E2 17523.317} C_VEL
LIN {X 0,Y 380.605,Z 940.24,A -85,B 0,C 180,E1 17521.95,E2 17521.95} C_VEL
LIN {X 0,Y 382.498,Z 922.717,A -85,B 0,C 180,E1 17520.861,E2 17520.861} C_VEL
LIN {X 0,Y 384.151,Z 904.146,A -85,B 0,C 180,E1 17520.024,E2 17520.024} C_VEL
LIN {X 0,Y 385.217,Z 885.396,A -85,B 0,C 180,E1 17519.467,E2 17519.467} C_VEL
LIN {X 0,Y 389.003,Z 720.871,A -85,B 0,C 180,E1 17516.344,E2 17516.344} C_VEL
LIN {X 0,Y 386.213,Z 694.763,A -85,B 0,C 180,E1 17515.473,E2 17515.473} C_VEL
LIN {X 0,Y 390.642,Z 664.867,A -85,B 0,C 180,E1 17512.1,E2 17512.1} C_VEL
LIN {X 0,Y 386.132,Z 650.372,A -85,B 0,C 180,E1 17509.578,E2 17509.578} C_VEL
LIN {X 0,Y 380.766,Z 635.757,A -85,B 0,C 180,E1 17506.667,E2 17506.667} C_VEL
LIN {X 0,Y 375,Z 621.766,A -85,B 0,C 180,E1 17503.464,E2 17503.464} C_VEL
LIN {X 0,Y 371.143,Z 613.419,A -85,B 0,C 180,E1 17501.269,E2 17501.269} C_VEL
LIN {X 0,Y 369.741,Z 609.889,A -85,B 0,C 180,E1 17500.233,E2 17500.233} C_VEL
LIN {X 0,Y 369.706,Z 609.739,A -85,B 0,C 180,E1 17496.3,E2 17496.3} C_VEL
LIN {X 0,Y 369.699,Z 609.734,A -85,B 0,C 180,E1 17492.377,E2 17492.377} C_VEL
LIN {X 0,Y 369.697,Z 609.732,A -85,B 0,C 180,E1 17488.424,E2 17488.424} C_VEL
LIN {X 0,Y 369.699,Z 609.731,A -85,B 0,C 180,E1 17484.273,E2 17484.273} C_VEL
LIN {X 0,Y 369.702,Z 609.735,A -85,B 0,C 180,E1 17480.205,E2 17480.205} C_VEL
LIN {X 0,Y 369.706,Z 609.742,A -85,B 0,C 180,E1 17476.174,E2 17476.174} C_VEL
LIN {X 0,Y 369.715,Z 609.745,A -85,B 0,C 180,E1 17472.177,E2 17472.177} C_VEL
LIN {X 0,Y 369.719,Z 609.731,A -85,B 0,C 180,E1 17468.084,E2 17468.084} C_VEL
LIN {X 0,Y 369.732,Z 609.72,A -85,B 0,C 180,E1 17464.187,E2 17464.187} C_VEL
LIN {X 0,Y 369.752,Z 609.719,A -85,B 0,C 180,E1 17460.155,E2 17460.155} C_VEL
LIN {X 0,Y 369.739,Z 609.724,A -85,B 0,C 180,E1 17455.968,E2 17455.968} C_VEL
LIN {X 0,Y 369.752,Z 609.729,A -85,B 0,C 180,E1 17451.916,E2 17451.916} C_VEL
LIN {X 0,Y 369.746,Z 609.73,A -85,B 0,C 180,E1 17447.664,E2 17447.664} C_VEL
LIN {X 0,Y 369.748,Z 609.731,A -85,B 0,C 180,E1 17443.666,E2 17443.666} C_VEL
LIN {X 0,Y 369.747,Z 609.728,A -85,B 0,C 180,E1 17439.583,E2 17439.583} C_VEL
LIN {X 0,Y 369.739,Z 609.73,A -85,B 0,C 180,E1 17435.559,E2 17435.559} C_VEL
LIN {X 0,Y 369.8,Z 610.135,A -85,B 0,C 180,E1 17434.881,E2 17434.881} C_VEL
LIN {X 0,Y 374.092,Z 621.055,A -85,B 0,C 180,E1 17431.563,E2 17431.563} C_VEL
LIN {X 0,Y 378.397,Z 633.213,A -85,B 0,C 180,E1 17428.275,E2 17428.275} C_VEL
LIN {X 0,Y 382.426,Z 646.431,A -85,B 0,C 180,E1 17425.069,E2 17425.069} C_VEL
LIN {X 0,Y 385.565,Z 659.172,A -85,B 0,C 180,E1 17422.265,E2 17422.265} C_VEL
LIN {X 0,Y 381.866,Z 685.087,A -85,B 0,C 180,E1 17418.04,E2 17418.04} C_VEL
LIN {X 0,Y 379.233,Z 706.555,A -85,B 0,C 180,E1 17414.613,E2 17414.613} C_VEL
LIN {X 0,Y 380.942,Z 715.292,A -85,B 0,C 180,E1 17414.189,E2 17414.189} C_VEL
LIN {X 0,Y 385.332,Z 739.069,A -85,B 0,C 180,E1 17413.241,E2 17413.241} C_VEL
LIN {X 0,Y 382.648,Z 833.89,A -85,B 0,C 180,E1 17411.271,E2 17411.271} C_VEL
LIN {X 0,Y 381.917,Z 849.936,A -85,B 0,C 180,E1 17410.656,E2 17410.656} C_VEL
LIN {X 0,Y 380.887,Z 864.47,A -85,B 0,C 180,E1 17409.83,E2 17409.83} C_VEL
LIN {X 0,Y 379.432,Z 879.576,A -85,B 0,C 180,E1 17408.648,E2 17408.648} C_VEL
LIN {X 0,Y 377.866,Z 892.627,A -85,B 0,C 180,E1 17407.297,E2 17407.297} C_VEL
LIN {X 0,Y 376.199,Z 904.819,A -85,B 0,C 180,E1 17405.688,E2 17405.688} C_VEL
LIN {X 0,Y 374.589,Z 915.451,A -85,B 0,C 180,E1 17403.888,E2 17403.888} C_VEL
LIN {X 0,Y 373.191,Z 924.134,A -85,B 0,C 180,E1 17402.038,E2 17402.038} C_VEL
LIN {X 0,Y 371.854,Z 932.085,A -85,B 0,C 180,E1 17399.83,E2 17399.83} C_VEL
LIN {X 0,Y 370.883,Z 937.979,A -85,B 0,C 180,E1 17397.625,E2 17397.625} C_VEL
LIN {X 0,Y 370.135,Z 942.57,A -85,B 0,C 180,E1 17395.094,E2 17395.094} C_VEL
LIN {X 0,Y 369.732,Z 944.948,A -85,B 0,C 180,E1 17392.75,E2 17392.75} C_VEL
LIN {X 0,Y 369.546,Z 945.708,A -85,B 0,C 180,E1 17390.262,E2 17390.262} C_VEL
LIN {X 0,Y 369.558,Z 944.586,A -85,B 0,C 180,E1 17387.756,E2 17387.756} C_VEL
LIN {X 0,Y 369.782,Z 941.788,A -85,B 0,C 180,E1 17385.366,E2 17385.366} C_VEL
LIN {X 0,Y 370.281,Z 936.893,A -85,B 0,C 180,E1 17382.888,E2 17382.888} C_VEL
LIN {X 0,Y 370.988,Z 930.735,A -85,B 0,C 180,E1 17380.717,E2 17380.717} C_VEL
LIN {X 0,Y 371.948,Z 923.012,A -85,B 0,C 180,E1 17378.658,E2 17378.658} C_VEL
LIN {X 0,Y 373.083,Z 913.906,A -85,B 0,C 180,E1 17376.772,E2 17376.772} C_VEL
LIN {X 0,Y 374.376,Z 903.122,A -85,B 0,C 180,E1 17375.001,E2 17375.001} C_VEL
LIN {X 0,Y 375.643,Z 891.368,A -85,B 0,C 180,E1 17373.48,E2 17373.48} C_VEL
LIN {X 0,Y 376.967,Z 878.1,A -85,B 0,C 180,E1 17372.128,E2 17372.128} C_VEL
LIN {X 0,Y 378.145,Z 863.261,A -85,B 0,C 180,E1 17370.984,E2 17370.984} C_VEL
LIN {X 0,Y 379.033,Z 848.292,A -85,B 0,C 180,E1 17370.146,E2 17370.146} C_VEL
LIN {X 0,Y 379.283,Z 842.821,A -85,B 0,C 180,E1 17369.91,E2 17369.91} C_VEL
LIN {X 0,Y 378.892,Z 836.415,A -85,B 0,C 180,E1 17369.637,E2 17369.637} C_VEL
LIN {X 0,Y 375.167,Z 822.95,A -85,B 0,C 180,E1 17369.024,E2 17369.024} C_VEL
LIN {X 0,Y 373.007,Z 813.436,A -85,B 0,C 180,E1 17368.674,E2 17368.674} C_VEL
LIN {X 0,Y 372.8,Z 809.066,A -85,B 0,C 180,E1 17368.565,E2 17368.565} C_VEL
LIN {X 0,Y 374.327,Z 737.276,A -85,B 0,C 180,E1 17367.121,E2 17367.121} C_VEL
LIN {X 0,Y 369.17,Z 706.902,A -85,B 0,C 180,E1 17366.078,E2 17366.078} C_VEL
LIN {X 0,Y 372.036,Z 679.692,A -85,B 0,C 180,E1 17361.811,E2 17361.811} C_VEL
LIN {X 0,Y 374.908,Z 655.85,A -85,B 0,C 180,E1 17357.993,E2 17357.993} C_VEL
LIN {X 0,Y 370.399,Z 638.63,A -85,B 0,C 180,E1 17354.514,E2 17354.514} C_VEL
LIN {X 0,Y 365.362,Z 621.683,A -85,B 0,C 180,E1 17350.828,E2 17350.828} C_VEL
LIN {X 0,Y 361.831,Z 610.85,A -85,B 0,C 180,E1 17348.243,E2 17348.243} C_VEL
LIN {X 0,Y 361.803,Z 610.703,A -85,B 0,C 180,E1 17344.11,E2 17344.11} C_VEL
LIN {X 0,Y 361.807,Z 610.669,A -85,B 0,C 180,E1 17339.986,E2 17339.986} C_VEL
LIN {X 0,Y 361.804,Z 610.725,A -85,B 0,C 180,E1 17335.721,E2 17335.721} C_VEL
LIN {X 0,Y 361.806,Z 610.718,A -85,B 0,C 180,E1 17331.452,E2 17331.452} C_VEL
LIN {X 0,Y 361.799,Z 610.706,A -85,B 0,C 180,E1 17327.317,E2 17327.317} C_VEL
LIN {X 0,Y 361.801,Z 610.726,A -85,B 0,C 180,E1 17323.148,E2 17323.148} C_VEL
LIN {X 0,Y 361.812,Z 610.718,A -85,B 0,C 180,E1 17319.055,E2 17319.055} C_VEL
LIN {X 0,Y 361.8,Z 610.705,A -85,B 0,C 180,E1 17314.836,E2 17314.836} C_VEL
LIN {X 0,Y 361.813,Z 610.727,A -85,B 0,C 180,E1 17310.745,E2 17310.745} C_VEL
LIN {X 0,Y 361.802,Z 610.694,A -85,B 0,C 180,E1 17306.596,E2 17306.596} C_VEL
LIN {X 0,Y 361.811,Z 610.727,A -85,B 0,C 180,E1 17302.418,E2 17302.418} C_VEL
LIN {X 0,Y 361.795,Z 610.692,A -85,B 0,C 180,E1 17298.198,E2 17298.198} C_VEL
LIN {X 0,Y 361.806,Z 610.727,A -85,B 0,C 180,E1 17294.068,E2 17294.068} C_VEL
LIN {X 0,Y 361.794,Z 610.696,A -85,B 0,C 180,E1 17289.866,E2 17289.866} C_VEL
LIN {X 0,Y 361.804,Z 610.725,A -85,B 0,C 180,E1 17285.798,E2 17285.798} C_VEL
LIN {X 0,Y 361.797,Z 610.698,A -85,B 0,C 180,E1 17281.584,E2 17281.584} C_VEL
LIN {X 0,Y 361.801,Z 610.729,A -85,B 0,C 180,E1 17277.466,E2 17277.466} C_VEL
LIN {X 0,Y 361.806,Z 610.696,A -85,B 0,C 180,E1 17273.335,E2 17273.335} C_VEL
LIN {X 0,Y 361.8,Z 610.73,A -85,B 0,C 180,E1 17269.169,E2 17269.169} C_VEL
LIN {X 0,Y 361.812,Z 610.702,A -85,B 0,C 180,E1 17265.108,E2 17265.108} C_VEL
LIN {X 0,Y 361.806,Z 610.72,A -85,B 0,C 180,E1 17260.933,E2 17260.933} C_VEL
LIN {X 0,Y 361.807,Z 610.73,A -85,B 0,C 180,E1 17256.723,E2 17256.723} C_VEL
LIN {X 0,Y 361.806,Z 610.72,A -85,B 0,C 180,E1 17252.511,E2 17252.511} C_VEL
LIN {X 0,Y 361.81,Z 610.714,A -85,B 0,C 180,E1 17248.514,E2 17248.514} C_VEL
LIN {X 0,Y 361.801,Z 610.719,A -85,B 0,C 180,E1 17244.331,E2 17244.331} C_VEL
LIN {X 0,Y 361.814,Z 610.728,A -85,B 0,C 180,E1 17240.125,E2 17240.125} C_VEL
LIN {X 0,Y 361.789,Z 610.939,A -85,B 0,C 180,E1 17236.951,E2 17236.951} C_VEL
LIN {X 0,Y 368.026,Z 627.459,A -85,B 0,C 180,E1 17233.725,E2 17233.725} C_VEL
LIN {X 0,Y 374.649,Z 646.117,A -85,B 0,C 180,E1 17230.483,E2 17230.483} C_VEL
LIN {X 0,Y 380.603,Z 664.495,A -85,B 0,C 180,E1 17227.576,E2 17227.576} C_VEL
LIN {X 0,Y 376.603,Z 695.037,A -85,B 0,C 180,E1 17224.248,E2 17224.248} C_VEL
LIN {X 0,Y 379.494,Z 724.355,A -85,B 0,C 180,E1 17223.421,E2 17223.421} C_VEL
LIN {X 0,Y 375.849,Z 889.452,A -85,B 0,C 180,E1 17220.307,E2 17220.307} C_VEL
LIN {X 0,Y 374.741,Z 907.988,A -85,B 0,C 180,E1 17219.694,E2 17219.694} C_VEL
LIN {X 0,Y 373.226,Z 925.777,A -85,B 0,C 180,E1 17218.831,E2 17218.831} C_VEL
LIN {X 0,Y 371.396,Z 943.591,A -85,B 0,C 180,E1 17217.66,E2 17217.66} C_VEL
LIN {X 0,Y 369.481,Z 960.126,A -85,B 0,C 180,E1 17216.261,E2 17216.261} C_VEL
LIN {X 0,Y 367.465,Z 975.868,A -85,B 0,C 180,E1 17214.602,E2 17214.602} C_VEL
LIN {X 0,Y 365.583,Z 990.677,A -85,B 0,C 180,E1 17212.683,E2 17212.683} C_VEL
LIN {X 0,Y 363.925,Z 1003.948,A -85,B 0,C 180,E1 17210.59,E2 17210.59} C_VEL
LIN {X 0,Y 362.484,Z 1016.556,A -85,B 0,C 180,E1 17208.162,E2 17208.162} C_VEL
LIN {X 0,Y 361.514,Z 1026.931,A -85,B 0,C 180,E1 17205.727,E2 17205.727} C_VEL
LIN {X 0,Y 360.931,Z 1035.902,A -85,B 0,C 180,E1 17203.13,E2 17203.13} C_VEL
LIN {X 0,Y 360.715,Z 1043.398,A -85,B 0,C 180,E1 17200.38,E2 17200.38} C_VEL
LIN {X 0,Y 360.795,Z 1049.027,A -85,B 0,C 180,E1 17197.645,E2 17197.645} C_VEL
LIN {X 0,Y 361.005,Z 1052.912,A -85,B 0,C 180,E1 17194.926,E2 17194.926} C_VEL
LIN {X 0,Y 361.199,Z 1055.128,A -85,B 0,C 180,E1 17192.221,E2 17192.221} C_VEL
LIN {X 0,Y 361.252,Z 1055.716,A -85,B 0,C 180,E1 17189.525,E2 17189.525} C_VEL
LIN {X 0,Y 361.118,Z 1054.686,A -85,B 0,C 180,E1 17186.826,E2 17186.826} C_VEL
LIN {X 0,Y 360.888,Z 1051.957,A -85,B 0,C 180,E1 17184.057,E2 17184.057} C_VEL
LIN {X 0,Y 360.692,Z 1047.418,A -85,B 0,C 180,E1 17181.231,E2 17181.231} C_VEL
LIN {X 0,Y 360.706,Z 1041.281,A -85,B 0,C 180,E1 17178.488,E2 17178.488} C_VEL
LIN {X 0,Y 361.1,Z 1033.262,A -85,B 0,C 180,E1 17175.725,E2 17175.725} C_VEL
LIN {X 0,Y 361.891,Z 1023.879,A -85,B 0,C 180,E1 17173.136,E2 17173.136} C_VEL
LIN {X 0,Y 363.224,Z 1012.313,A -85,B 0,C 180,E1 17170.544,E2 17170.544} C_VEL
LIN {X 0,Y 364.993,Z 999.107,A -85,B 0,C 180,E1 17168.127,E2 17168.127} C_VEL
LIN {X 0,Y 366.977,Z 985.286,A -85,B 0,C 180,E1 17166.049,E2 17166.049} C_VEL
LIN {X 0,Y 369.14,Z 970.581,A -85,B 0,C 180,E1 17164.232,E2 17164.232} C_VEL
LIN {X 0,Y 371.461,Z 954.283,A -85,B 0,C 180,E1 17162.595,E2 17162.595} C_VEL
LIN {X 0,Y 373.561,Z 937.925,A -85,B 0,C 180,E1 17161.286,E2 17161.286} C_VEL
LIN {X 0,Y 375.562,Z 920.164,A -85,B 0,C 180,E1 17160.195,E2 17160.195} C_VEL
LIN {X 0,Y 377.186,Z 902.108,A -85,B 0,C 180,E1 17159.394,E2 17159.394} C_VEL
LIN {X 0,Y 378.244,Z 883.592,A -85,B 0,C 180,E1 17158.852,E2 17158.852} C_VEL
LIN {X 0,Y 382.193,Z 721.907,A -85,B 0,C 180,E1 17155.735,E2 17155.735} C_VEL
LIN {X 0,Y 379.341,Z 694.933,A -85,B 0,C 180,E1 17154.81,E2 17154.81} C_VEL
LIN {X 0,Y 383.601,Z 667.803,A -85,B 0,C 180,E1 17151.68,E2 17151.68} C_VEL
LIN {X 0,Y 379.087,Z 653.394,A -85,B 0,C 180,E1 17149.082,E2 17149.082} C_VEL
LIN {X 0,Y 374.307,Z 640.133,A -85,B 0,C 180,E1 17146.377,E2 17146.377} C_VEL
LIN {X 0,Y 368.662,Z 626.404,A -85,B 0,C 180,E1 17143.15,E2 17143.15} C_VEL
LIN {X 0,Y 364.868,Z 618.131,A -85,B 0,C 180,E1 17140.915,E2 17140.915} C_VEL
LIN {X 0,Y 362.98,Z 614.001,A -85,B 0,C 180,E1 17139.722,E2 17139.722} C_VEL
LIN {X 0,Y 361.775,Z 610.878,A -85,B 0,C 180,E1 17138.727,E2 17138.727} C_VEL
LIN {X 0,Y 361.758,Z 610.723,A -85,B 0,C 180,E1 17134.549,E2 17134.549} C_VEL
LIN {X 0,Y 361.759,Z 610.728,A -85,B 0,C 180,E1 17130.384,E2 17130.384} C_VEL
LIN {X 0,Y 361.764,Z 610.729,A -85,B 0,C 180,E1 17126.245,E2 17126.245} C_VEL
LIN {X 0,Y 361.76,Z 610.727,A -85,B 0,C 180,E1 17122.079,E2 17122.079} C_VEL
LIN {X 0,Y 361.764,Z 610.721,A -85,B 0,C 180,E1 17117.865,E2 17117.865} C_VEL
LIN {X 0,Y 361.762,Z 610.714,A -85,B 0,C 180,E1 17113.75,E2 17113.75} C_VEL
LIN {X 0,Y 361.766,Z 610.709,A -85,B 0,C 180,E1 17109.545,E2 17109.545} C_VEL
LIN {X 0,Y 361.766,Z 610.715,A -85,B 0,C 180,E1 17105.392,E2 17105.392} C_VEL
LIN {X 0,Y 361.768,Z 610.727,A -85,B 0,C 180,E1 17101.267,E2 17101.267} C_VEL
LIN {X 0,Y 361.772,Z 610.733,A -85,B 0,C 180,E1 17097.148,E2 17097.148} C_VEL
LIN {X 0,Y 361.772,Z 610.735,A -85,B 0,C 180,E1 17093.015,E2 17093.015} C_VEL
LIN {X 0,Y 361.776,Z 610.734,A -85,B 0,C 180,E1 17088.845,E2 17088.845} C_VEL
LIN {X 0,Y 361.775,Z 610.735,A -85,B 0,C 180,E1 17084.614,E2 17084.614} C_VEL
LIN {X 0,Y 361.779,Z 610.73,A -85,B 0,C 180,E1 17080.463,E2 17080.463} C_VEL
LIN {X 0,Y 361.808,Z 610.925,A -85,B 0,C 180,E1 17076.42,E2 17076.42} C_VEL
LIN {X 0,Y 366.168,Z 621.768,A -85,B 0,C 180,E1 17072.87,E2 17072.87} C_VEL
LIN {X 0,Y 370.613,Z 634.125,A -85,B 0,C 180,E1 17069.343,E2 17069.343} C_VEL
LIN {X 0,Y 374.584,Z 646.884,A -85,B 0,C 180,E1 17066.091,E2 17066.091} C_VEL
LIN {X 0,Y 377.956,Z 659.926,A -85,B 0,C 180,E1 17063.093,E2 17063.093} C_VEL
LIN {X 0,Y 378.407,Z 662.373,A -85,B 0,C 180,E1 17062.574,E2 17062.574} C_VEL
LIN {X 0,Y 374.374,Z 689.326,A -85,B 0,C 180,E1 17058.111,E2 17058.111} C_VEL
LIN {X 0,Y 372.162,Z 706.536,A -85,B 0,C 180,E1 17055.326,E2 17055.326} C_VEL
LIN {X 0,Y 377.343,Z 732.921,A -85,B 0,C 180,E1 17054.137,E2 17054.137} C_VEL
LIN {X 0,Y 378.488,Z 741.112,A -85,B 0,C 180,E1 17053.84,E2 17053.84} C_VEL
LIN {X 0,Y 375.697,Z 834.601,A -85,B 0,C 180,E1 17051.86,E2 17051.86} C_VEL
LIN {X 0,Y 374.919,Z 850.746,A -85,B 0,C 180,E1 17051.231,E2 17051.231} C_VEL
LIN {X 0,Y 373.852,Z 865.07,A -85,B 0,C 180,E1 17050.405,E2 17050.405} C_VEL
LIN {X 0,Y 372.341,Z 879.958,A -85,B 0,C 180,E1 17049.227,E2 17049.227} C_VEL
LIN {X 0,Y 370.716,Z 892.905,A -85,B 0,C 180,E1 17047.883,E2 17047.883} C_VEL
LIN {X 0,Y 368.906,Z 905.431,A -85,B 0,C 180,E1 17046.217,E2 17046.217} C_VEL
LIN {X 0,Y 367.206,Z 916.034,A -85,B 0,C 180,E1 17044.407,E2 17044.407} C_VEL
LIN {X 0,Y 365.616,Z 925.275,A -85,B 0,C 180,E1 17042.412,E2 17042.412} C_VEL
LIN {X 0,Y 364.16,Z 933.306,A -85,B 0,C 180,E1 17040.13,E2 17040.13} C_VEL
LIN {X 0,Y 363.11,Z 939.168,A -85,B 0,C 180,E1 17037.882,E2 17037.882} C_VEL
LIN {X 0,Y 362.302,Z 943.707,A -85,B 0,C 180,E1 17035.325,E2 17035.325} C_VEL
LIN {X 0,Y 361.854,Z 946.118,A -85,B 0,C 180,E1 17032.93,E2 17032.93} C_VEL
LIN {X 0,Y 361.64,Z 946.908,A -85,B 0,C 180,E1 17030.387,E2 17030.387} C_VEL
LIN {X 0,Y 361.639,Z 945.869,A -85,B 0,C 180,E1 17027.872,E2 17027.872} C_VEL
LIN {X 0,Y 361.874,Z 943.057,A -85,B 0,C 180,E1 17025.357,E2 17025.357} C_VEL
LIN {X 0,Y 362.363,Z 938.398,A -85,B 0,C 180,E1 17022.915,E2 17022.915} C_VEL
LIN {X 0,Y 363.117,Z 932.186,A -85,B 0,C 180,E1 17020.631,E2 17020.631} C_VEL
LIN {X 0,Y 364.202,Z 923.885,A -85,B 0,C 180,E1 17018.366,E2 17018.366} C_VEL
LIN {X 0,Y 365.399,Z 914.714,A -85,B 0,C 180,E1 17016.441,E2 17016.441} C_VEL
LIN {X 0,Y 366.779,Z 903.731,A -85,B 0,C 180,E1 17014.612,E2 17014.612} C_VEL
LIN {X 0,Y 368.213,Z 890.979,A -85,B 0,C 180,E1 17012.957,E2 17012.957} C_VEL
LIN {X 0,Y 369.543,Z 877.995,A -85,B 0,C 180,E1 17011.641,E2 17011.641} C_VEL
LIN {X 0,Y 370.802,Z 862.722,A -85,B 0,C 180,E1 17010.463,E2 17010.463} C_VEL
LIN {X 0,Y 371.723,Z 847.022,A -85,B 0,C 180,E1 17009.605,E2 17009.605} C_VEL
LIN {X 0,Y 372.293,Z 831.438,A -85,B 0,C 180,E1 17009.048,E2 17009.048} C_VEL
LIN {X 0,Y 372.8,Z 809.066,A -85,B 0,C 180,E1 17008.565,E2 17008.565} C_VEL
LIN {X 0,Y 372.11,Z 801.461,A -85,B 0,C 180,E1 17008.349,E2 17008.349} C_VEL
LIN {X 0,Y 366.873,Z 781.519,A -85,B 0,C 180,E1 17007.55,E2 17007.55} C_VEL
LIN {X 0,Y 366.342,Z 774.982,A -85,B 0,C 180,E1 17007.368,E2 17007.368} C_VEL
LIN {X 0,Y 367.038,Z 738.309,A -85,B 0,C 180,E1 17006.618,E2 17006.618} C_VEL
LIN {X 0,Y 361.722,Z 706.454,A -85,B 0,C 180,E1 17005.481,E2 17005.481} C_VEL
LIN {X 0,Y 364.885,Z 678.638,A -85,B 0,C 180,E1 17001.014,E2 17001.014} C_VEL
LIN {X 0,Y 367.417,Z 658.166,A -85,B 0,C 180,E1 16997.678,E2 16997.678} C_VEL
LIN {X 0,Y 363.013,Z 641.193,A -85,B 0,C 180,E1 16994.176,E2 16994.176} C_VEL
LIN {X 0,Y 358.25,Z 625.122,A -85,B 0,C 180,E1 16990.602,E2 16990.602} C_VEL
LIN {X 0,Y 353.874,Z 611.831,A -85,B 0,C 180,E1 16987.358,E2 16987.358} C_VEL
LIN {X 0,Y 353.859,Z 611.72,A -85,B 0,C 180,E1 16983.121,E2 16983.121} C_VEL
LIN {X 0,Y 353.851,Z 611.652,A -85,B 0,C 180,E1 16978.89,E2 16978.89} C_VEL
LIN {X 0,Y 353.858,Z 611.723,A -85,B 0,C 180,E1 16974.746,E2 16974.746} C_VEL
LIN {X 0,Y 353.859,Z 611.718,A -85,B 0,C 180,E1 16970.479,E2 16970.479} C_VEL
LIN {X 0,Y 353.855,Z 611.697,A -85,B 0,C 180,E1 16966.333,E2 16966.333} C_VEL
LIN {X 0,Y 353.852,Z 611.701,A -85,B 0,C 180,E1 16962.241,E2 16962.241} C_VEL
LIN {X 0,Y 353.852,Z 611.717,A -85,B 0,C 180,E1 16958.024,E2 16958.024} C_VEL
LIN {X 0,Y 353.849,Z 611.686,A -85,B 0,C 180,E1 16953.823,E2 16953.823} C_VEL
LIN {X 0,Y 353.852,Z 611.722,A -85,B 0,C 180,E1 16949.636,E2 16949.636} C_VEL
LIN {X 0,Y 353.847,Z 611.682,A -85,B 0,C 180,E1 16945.436,E2 16945.436} C_VEL
LIN {X 0,Y 353.847,Z 611.722,A -85,B 0,C 180,E1 16941.378,E2 16941.378} C_VEL
LIN {X 0,Y 353.838,Z 611.679,A -85,B 0,C 180,E1 16937.231,E2 16937.231} C_VEL
LIN {X 0,Y 353.841,Z 611.722,A -85,B 0,C 180,E1 16933.066,E2 16933.066} C_VEL
LIN {X 0,Y 353.834,Z 611.679,A -85,B 0,C 180,E1 16928.941,E2 16928.941} C_VEL
LIN {X 0,Y 353.836,Z 611.719,A -85,B 0,C 180,E1 16924.863,E2 16924.863} C_VEL
LIN {X 0,Y 353.827,Z 611.683,A -85,B 0,C 180,E1 16920.648,E2 16920.648} C_VEL
LIN {X 0,Y 353.835,Z 611.722,A -85,B 0,C 180,E1 16916.436,E2 16916.436} C_VEL
LIN {X 0,Y 353.824,Z 611.687,A -85,B 0,C 180,E1 16912.368,E2 16912.368} C_VEL
LIN {X 0,Y 353.829,Z 611.723,A -85,B 0,C 180,E1 16908.261,E2 16908.261} C_VEL
LIN {X 0,Y 353.825,Z 611.709,A -85,B 0,C 180,E1 16904.091,E2 16904.091} C_VEL
LIN {X 0,Y 353.826,Z 611.703,A -85,B 0,C 180,E1 16900.006,E2 16900.006} C_VEL
LIN {X 0,Y 353.826,Z 611.723,A -85,B 0,C 180,E1 16895.811,E2 16895.811} C_VEL
LIN {X 0,Y 353.824,Z 611.723,A -85,B 0,C 180,E1 16891.658,E2 16891.658} C_VEL
LIN {X 0,Y 353.824,Z 611.721,A -85,B 0,C 180,E1 16887.526,E2 16887.526} C_VEL
LIN {X 0,Y 353.823,Z 611.726,A -85,B 0,C 180,E1 16883.375,E2 16883.375} C_VEL
LIN {X 0,Y 353.822,Z 611.721,A -85,B 0,C 180,E1 16879.231,E2 16879.231} C_VEL
LIN {X 0,Y 353.899,Z 612.043,A -85,B 0,C 180,E1 16877.823,E2 16877.823} C_VEL
LIN {X 0,Y 360.463,Z 629.372,A -85,B 0,C 180,E1 16874.348,E2 16874.348} C_VEL
LIN {X 0,Y 366.444,Z 646.139,A -85,B 0,C 180,E1 16871.324,E2 16871.324} C_VEL
LIN {X 0,Y 373.082,Z 666.461,A -85,B 0,C 180,E1 16868.009,E2 16868.009} C_VEL
LIN {X 0,Y 369.333,Z 694.98,A -85,B 0,C 180,E1 16864.802,E2 16864.802} C_VEL
LIN {X 0,Y 372.237,Z 725.29,A -85,B 0,C 180,E1 16863.925,E2 16863.925} C_VEL
LIN {X 0,Y 368.476,Z 888.817,A -85,B 0,C 180,E1 16860.792,E2 16860.792} C_VEL
LIN {X 0,Y 367.337,Z 907.381,A -85,B 0,C 180,E1 16860.168,E2 16860.168} C_VEL
LIN {X 0,Y 365.704,Z 925.746,A -85,B 0,C 180,E1 16859.257,E2 16859.257} C_VEL
LIN {X 0,Y 363.884,Z 942.751,A -85,B 0,C 180,E1 16858.113,E2 16858.113} C_VEL
LIN {X 0,Y 361.877,Z 959.368,A -85,B 0,C 180,E1 16856.679,E2 16856.679} C_VEL
LIN {X 0,Y 359.781,Z 975.081,A -85,B 0,C 180,E1 16854.988,E2 16854.988} C_VEL
LIN {X 0,Y 357.817,Z 989.855,A -85,B 0,C 180,E1 16853.03,E2 16853.03} C_VEL
LIN {X 0,Y 356.088,Z 1003.084,A -85,B 0,C 180,E1 16850.892,E2 16850.892} C_VEL
LIN {X 0,Y 354.584,Z 1015.657,A -85,B 0,C 180,E1 16848.411,E2 16848.411} C_VEL
LIN {X 0,Y 353.571,Z 1025.997,A -85,B 0,C 180,E1 16845.921,E2 16845.921} C_VEL
LIN {X 0,Y 352.971,Z 1034.946,A -85,B 0,C 180,E1 16843.265,E2 16843.265} C_VEL
LIN {X 0,Y 352.752,Z 1042.519,A -85,B 0,C 180,E1 16840.406,E2 16840.406} C_VEL
LIN {X 0,Y 352.862,Z 1048.278,A -85,B 0,C 180,E1 16837.49,E2 16837.49} C_VEL
LIN {X 0,Y 353.102,Z 1052.086,A -85,B 0,C 180,E1 16834.632,E2 16834.632} C_VEL
LIN {X 0,Y 353.304,Z 1054.055,A -85,B 0,C 180,E1 16831.946,E2 16831.946} C_VEL
LIN {X 0,Y 353.337,Z 1054.466,A -85,B 0,C 180,E1 16829.19,E2 16829.19} C_VEL
LIN {X 0,Y 353.168,Z 1053.248,A -85,B 0,C 180,E1 16826.429,E2 16826.429} C_VEL
LIN {X 0,Y 352.907,Z 1050.412,A -85,B 0,C 180,E1 16823.656,E2 16823.656} C_VEL
LIN {X 0,Y 352.713,Z 1045.921,A -85,B 0,C 180,E1 16820.866,E2 16820.866} C_VEL
LIN {X 0,Y 352.751,Z 1039.69,A -85,B 0,C 180,E1 16818.059,E2 16818.059} C_VEL
LIN {X 0,Y 353.21,Z 1031.586,A -85,B 0,C 180,E1 16815.24,E2 16815.24} C_VEL
LIN {X 0,Y 354.107,Z 1022.047,A -85,B 0,C 180,E1 16812.585,E2 16812.585} C_VEL
LIN {X 0,Y 355.579,Z 1010.333,A -85,B 0,C 180,E1 16809.937,E2 16809.937} C_VEL
LIN {X 0,Y 357.366,Z 997.919,A -85,B 0,C 180,E1 16807.635,E2 16807.635} C_VEL
LIN {X 0,Y 359.477,Z 984.121,A -85,B 0,C 180,E1 16805.517,E2 16805.517} C_VEL
LIN {X 0,Y 361.75,Z 969.611,A -85,B 0,C 180,E1 16803.687,E2 16803.687} C_VEL
LIN {X 0,Y 364.102,Z 953.965,A -85,B 0,C 180,E1 16802.082,E2 16802.082} C_VEL
LIN {X 0,Y 366.302,Z 937.75,A -85,B 0,C 180,E1 16800.752,E2 16800.752} C_VEL
LIN {X 0,Y 368.414,Z 920.137,A -85,B 0,C 180,E1 16799.637,E2 16799.637} C_VEL
LIN {X 0,Y 370.147,Z 901.83,A -85,B 0,C 180,E1 16798.804,E2 16798.804} C_VEL
LIN {X 0,Y 371.269,Z 883.275,A -85,B 0,C 180,E1 16798.248,E2 16798.248} C_VEL
LIN {X 0,Y 375.419,Z 722.811,A -85,B 0,C 180,E1 16795.1,E2 16795.1} C_VEL
LIN {X 0,Y 372.527,Z 695.564,A -85,B 0,C 180,E1 16794.151,E2 16794.151} C_VEL
LIN {X 0,Y 376.674,Z 671.055,A -85,B 0,C 180,E1 16791.298,E2 16791.298} C_VEL
LIN {X 0,Y 372.103,Z 656.336,A -85,B 0,C 180,E1 16788.563,E2 16788.563} C_VEL
LIN {X 0,Y 367.243,Z 642.971,A -85,B 0,C 180,E1 16785.729,E2 16785.729} C_VEL
LIN {X 0,Y 362.239,Z 630.791,A -85,B 0,C 180,E1 16782.759,E2 16782.759} C_VEL
LIN {X 0,Y 358.876,Z 623.258,A -85,B 0,C 180,E1 16780.688,E2 16780.688} C_VEL
LIN {X 0,Y 357.028,Z 619.161,A -85,B 0,C 180,E1 16779.473,E2 16779.473} C_VEL
LIN {X 0,Y 355.165,Z 615.232,A -85,B 0,C 180,E1 16778.239,E2 16778.239} C_VEL
LIN {X 0,Y 353.843,Z 611.845,A -85,B 0,C 180,E1 16777.06,E2 16777.06} C_VEL
LIN {X 0,Y 353.837,Z 611.719,A -85,B 0,C 180,E1 16773.05,E2 16773.05} C_VEL
LIN {X 0,Y 353.852,Z 611.714,A -85,B 0,C 180,E1 16769.078,E2 16769.078} C_VEL
LIN {X 0,Y 353.847,Z 611.713,A -85,B 0,C 180,E1 16764.899,E2 16764.899} C_VEL
LIN {X 0,Y 353.857,Z 611.717,A -85,B 0,C 180,E1 16760.856,E2 16760.856} C_VEL
LIN {X 0,Y 353.857,Z 611.721,A -85,B 0,C 180,E1 16756.689,E2 16756.689} C_VEL
LIN {X 0,Y 353.858,Z 611.714,A -85,B 0,C 180,E1 16752.566,E2 16752.566} C_VEL
LIN {X 0,Y 353.853,Z 611.703,A -85,B 0,C 180,E1 16748.285,E2 16748.285} C_VEL
LIN {X 0,Y 353.853,Z 611.696,A -85,B 0,C 180,E1 16744.213,E2 16744.213} C_VEL
LIN {X 0,Y 353.863,Z 611.695,A -85,B 0,C 180,E1 16740,E2 16740} C_VEL
LIN {X 0,Y 353.854,Z 611.7,A -85,B 0,C 180,E1 16735.787,E2 16735.787} C_VEL
LIN {X 0,Y 353.866,Z 611.703,A -85,B 0,C 180,E1 16731.714,E2 16731.714} C_VEL
LIN {X 0,Y 353.86,Z 611.705,A -85,B 0,C 180,E1 16727.433,E2 16727.433} C_VEL
LIN {X 0,Y 353.863,Z 611.704,A -85,B 0,C 180,E1 16723.308,E2 16723.308} C_VEL
LIN {X 0,Y 353.868,Z 611.703,A -85,B 0,C 180,E1 16719.144,E2 16719.144} C_VEL
LIN {X 0,Y 353.892,Z 612.018,A -85,B 0,C 180,E1 16717.969,E2 16717.969} C_VEL
LIN {X 0,Y 357.464,Z 620.963,A -85,B 0,C 180,E1 16714.839,E2 16714.839} C_VEL
LIN {X 0,Y 360.922,Z 629.572,A -85,B 0,C 180,E1 16712.083,E2 16712.083} C_VEL
LIN {X 0,Y 365.086,Z 641.763,A -85,B 0,C 180,E1 16708.644,E2 16708.644} C_VEL
LIN {X 0,Y 368.727,Z 654.263,A -85,B 0,C 180,E1 16705.477,E2 16705.477} C_VEL
LIN {X 0,Y 371.306,Z 665.268,A -85,B 0,C 180,E1 16702.949,E2 16702.949} C_VEL
LIN {X 0,Y 367.044,Z 692.381,A -85,B 0,C 180,E1 16698.385,E2 16698.385} C_VEL
LIN {X 0,Y 365.144,Z 706.535,A -85,B 0,C 180,E1 16696.068,E2 16696.068} C_VEL
LIN {X 0,Y 371.016,Z 736.511,A -85,B 0,C 180,E1 16694.693,E2 16694.693} C_VEL
LIN {X 0,Y 371.733,Z 742.574,A -85,B 0,C 180,E1 16694.478,E2 16694.478} C_VEL
LIN {X 0,Y 368.793,Z 835.368,A -85,B 0,C 180,E1 16692.472,E2 16692.472} C_VEL
LIN {X 0,Y 367.96,Z 851.597,A -85,B 0,C 180,E1 16691.825,E2 16691.825} C_VEL
LIN {X 0,Y 366.81,Z 866.131,A -85,B 0,C 180,E1 16690.969,E2 16690.969} C_VEL
LIN {X 0,Y 365.181,Z 881.311,A -85,B 0,C 180,E1 16689.741,E2 16689.741} C_VEL
LIN {X 0,Y 363.46,Z 894.189,A -85,B 0,C 180,E1 16688.369,E2 16688.369} C_VEL
LIN {X 0,Y 361.555,Z 906.623,A -85,B 0,C 180,E1 16686.679,E2 16686.679} C_VEL
LIN {X 0,Y 359.666,Z 917.666,A -85,B 0,C 180,E1 16684.743,E2 16684.743} C_VEL
LIN {X 0,Y 358.058,Z 926.418,A -85,B 0,C 180,E1 16682.802,E2 16682.802} C_VEL
LIN {X 0,Y 356.516,Z 934.349,A -85,B 0,C 180,E1 16680.505,E2 16680.505} C_VEL
LIN {X 0,Y 355.374,Z 940.257,A -85,B 0,C 180,E1 16678.208,E2 16678.208} C_VEL
LIN {X 0,Y 354.476,Z 944.865,A -85,B 0,C 180,E1 16675.567,E2 16675.567} C_VEL
LIN {X 0,Y 353.981,Z 947.3,A -85,B 0,C 180,E1 16673.117,E2 16673.117} C_VEL
LIN {X 0,Y 353.735,Z 948.108,A -85,B 0,C 180,E1 16670.517,E2 16670.517} C_VEL
LIN {X 0,Y 353.724,Z 947.112,A -85,B 0,C 180,E1 16667.945,E2 16667.945} C_VEL
LIN {X 0,Y 353.955,Z 944.384,A -85,B 0,C 180,E1 16665.398,E2 16665.398} C_VEL
LIN {X 0,Y 354.462,Z 939.743,A -85,B 0,C 180,E1 16662.876,E2 16662.876} C_VEL
LIN {X 0,Y 355.245,Z 933.616,A -85,B 0,C 180,E1 16660.541,E2 16660.541} C_VEL
LIN {X 0,Y 356.364,Z 925.383,A -85,B 0,C 180,E1 16658.227,E2 16658.227} C_VEL
LIN {X 0,Y 357.607,Z 916.343,A -85,B 0,C 180,E1 16656.26,E2 16656.26} C_VEL
LIN {X 0,Y 359.103,Z 904.958,A -85,B 0,C 180,E1 16654.311,E2 16654.311} C_VEL
LIN {X 0,Y 360.598,Z 892.271,A -85,B 0,C 180,E1 16652.622,E2 16652.622} C_VEL
LIN {X 0,Y 362.035,Z 878.831,A -85,B 0,C 180,E1 16651.228,E2 16651.228} C_VEL
LIN {X 0,Y 363.287,Z 864.275,A -85,B 0,C 180,E1 16650.079,E2 16650.079} C_VEL
LIN {X 0,Y 364.245,Z 849.173,A -85,B 0,C 180,E1 16649.213,E2 16649.213} C_VEL
LIN {X 0,Y 364.894,Z 833.114,A -85,B 0,C 180,E1 16648.601,E2 16648.601} C_VEL
LIN {X 0,Y 366.342,Z 774.982,A -85,B 0,C 180,E1 16647.368,E2 16647.368} C_VEL
LIN {X 0,Y 365.627,Z 767.374,A -85,B 0,C 180,E1 16647.147,E2 16647.147} C_VEL
LIN {X 0,Y 360.464,Z 747.424,A -85,B 0,C 180,E1 16646.326,E2 16646.326} C_VEL
LIN {X 0,Y 359.973,Z 740.884,A -85,B 0,C 180,E1 16646.143,E2 16646.143} C_VEL
LIN {X 0,Y 354.31,Z 706.422,A -85,B 0,C 180,E1 16644.9,E2 16644.9} C_VEL
LIN {X 0,Y 357.653,Z 678.503,A -85,B 0,C 180,E1 16640.343,E2 16640.343} C_VEL
LIN {X 0,Y 359.894,Z 660.332,A -85,B 0,C 180,E1 16637.321,E2 16637.321} C_VEL
LIN {X 0,Y 355.64,Z 643.834,A -85,B 0,C 180,E1 16633.839,E2 16633.839} C_VEL
LIN {X 0,Y 350.991,Z 628.138,A -85,B 0,C 180,E1 16630.271,E2 16630.271} C_VEL
LIN {X 0,Y 346.488,Z 614.773,A -85,B 0,C 180,E1 16627.006,E2 16627.006} C_VEL
LIN {X 0,Y 345.936,Z 612.751,A -85,B 0,C 180,E1 16626.381,E2 16626.381} C_VEL
LIN {X 0,Y 345.933,Z 612.695,A -85,B 0,C 180,E1 16622.08,E2 16622.08} C_VEL
LIN {X 0,Y 345.921,Z 612.647,A -85,B 0,C 180,E1 16617.87,E2 16617.87} C_VEL
LIN {X 0,Y 345.925,Z 612.699,A -85,B 0,C 180,E1 16613.663,E2 16613.663} C_VEL
LIN {X 0,Y 345.935,Z 612.707,A -85,B 0,C 180,E1 16609.434,E2 16609.434} C_VEL
LIN {X 0,Y 345.922,Z 612.704,A -85,B 0,C 180,E1 16605.085,E2 16605.085} C_VEL
LIN {X 0,Y 345.913,Z 612.676,A -85,B 0,C 180,E1 16600.772,E2 16600.772} C_VEL
LIN {X 0,Y 345.912,Z 612.707,A -85,B 0,C 180,E1 16596.528,E2 16596.528} C_VEL
LIN {X 0,Y 345.907,Z 612.688,A -85,B 0,C 180,E1 16592.327,E2 16592.327} C_VEL
LIN {X 0,Y 345.908,Z 612.695,A -85,B 0,C 180,E1 16588.11,E2 16588.11} C_VEL
LIN {X 0,Y 345.902,Z 612.695,A -85,B 0,C 180,E1 16583.872,E2 16583.872} C_VEL
LIN {X 0,Y 345.9,Z 612.69,A -85,B 0,C 180,E1 16579.592,E2 16579.592} C_VEL
LIN {X 0,Y 345.899,Z 612.694,A -85,B 0,C 180,E1 16575.251,E2 16575.251} C_VEL
LIN {X 0,Y 345.899,Z 612.689,A -85,B 0,C 180,E1 16570.999,E2 16570.999} C_VEL
LIN {X 0,Y 345.899,Z 612.69,A -85,B 0,C 180,E1 16566.807,E2 16566.807} C_VEL
LIN {X 0,Y 345.898,Z 612.691,A -85,B 0,C 180,E1 16562.651,E2 16562.651} C_VEL
LIN {X 0,Y 345.892,Z 612.694,A -85,B 0,C 180,E1 16558.51,E2 16558.51} C_VEL
LIN {X 0,Y 345.891,Z 612.69,A -85,B 0,C 180,E1 16554.36,E2 16554.36} C_VEL
LIN {X 0,Y 345.893,Z 612.704,A -85,B 0,C 180,E1 16550.181,E2 16550.181} C_VEL
LIN {X 0,Y 345.885,Z 612.685,A -85,B 0,C 180,E1 16546.118,E2 16546.118} C_VEL
LIN {X 0,Y 345.89,Z 612.713,A -85,B 0,C 180,E1 16541.983,E2 16541.983} C_VEL
LIN {X 0,Y 345.884,Z 612.702,A -85,B 0,C 180,E1 16537.748,E2 16537.748} C_VEL
LIN {X 0,Y 345.887,Z 612.69,A -85,B 0,C 180,E1 16533.566,E2 16533.566} C_VEL
LIN {X 0,Y 345.881,Z 612.696,A -85,B 0,C 180,E1 16529.481,E2 16529.481} C_VEL
LIN {X 0,Y 345.883,Z 612.698,A -85,B 0,C 180,E1 16525.287,E2 16525.287} C_VEL
LIN {X 0,Y 345.88,Z 612.701,A -85,B 0,C 180,E1 16521.149,E2 16521.149} C_VEL
LIN {X 0,Y 345.921,Z 612.943,A -85,B 0,C 180,E1 16518.837,E2 16518.837} C_VEL
LIN {X 0,Y 352.252,Z 629.323,A -85,B 0,C 180,E1 16515.371,E2 16515.371} C_VEL
LIN {X 0,Y 358.817,Z 647.708,A -85,B 0,C 180,E1 16511.926,E2 16511.926} C_VEL
LIN {X 0,Y 365.441,Z 668.083,A -85,B 0,C 180,E1 16508.51,E2 16508.51} C_VEL
LIN {X 0,Y 365.777,Z 669.73,A -85,B 0,C 180,E1 16508.264,E2 16508.264} C_VEL
LIN {X 0,Y 362.106,Z 695.138,A -85,B 0,C 180,E1 16505.368,E2 16505.368} C_VEL
LIN {X 0,Y 365.007,Z 726.139,A -85,B 0,C 180,E1 16504.449,E2 16504.449} C_VEL
LIN {X 0,Y 361.104,Z 888.103,A -85,B 0,C 180,E1 16501.289,E2 16501.289} C_VEL
LIN {X 0,Y 359.945,Z 906.568,A -85,B 0,C 180,E1 16500.658,E2 16500.658} C_VEL
LIN {X 0,Y 358.264,Z 924.786,A -85,B 0,C 180,E1 16499.741,E2 16499.741} C_VEL
LIN {X 0,Y 356.388,Z 941.783,A -85,B 0,C 180,E1 16498.583,E2 16498.583} C_VEL
LIN {X 0,Y 354.292,Z 958.53,A -85,B 0,C 180,E1 16497.115,E2 16497.115} C_VEL
LIN {X 0,Y 352.116,Z 974.269,A -85,B 0,C 180,E1 16495.39,E2 16495.39} C_VEL
LIN {X 0,Y 350.066,Z 989.031,A -85,B 0,C 180,E1 16493.392,E2 16493.392} C_VEL
LIN {X 0,Y 348.259,Z 1002.218,A -85,B 0,C 180,E1 16491.208,E2 16491.208} C_VEL
LIN {X 0,Y 346.78,Z 1014.015,A -85,B 0,C 180,E1 16488.84,E2 16488.84} C_VEL
LIN {X 0,Y 345.652,Z 1024.843,A -85,B 0,C 180,E1 16486.185,E2 16486.185} C_VEL
LIN {X 0,Y 345.012,Z 1033.978,A -85,B 0,C 180,E1 16483.406,E2 16483.406} C_VEL
LIN {X 0,Y 344.793,Z 1041.408,A -85,B 0,C 180,E1 16480.527,E2 16480.527} C_VEL
LIN {X 0,Y 344.909,Z 1046.956,A -85,B 0,C 180,E1 16477.664,E2 16477.664} C_VEL
LIN {X 0,Y 345.167,Z 1050.746,A -85,B 0,C 180,E1 16474.813,E2 16474.813} C_VEL
LIN {X 0,Y 345.391,Z 1052.833,A -85,B 0,C 180,E1 16471.991,E2 16471.991} C_VEL
LIN {X 0,Y 345.425,Z 1053.274,A -85,B 0,C 180,E1 16469.171,E2 16469.171} C_VEL
LIN {X 0,Y 345.236,Z 1052.076,A -85,B 0,C 180,E1 16466.347,E2 16466.347} C_VEL
LIN {X 0,Y 344.944,Z 1049.25,A -85,B 0,C 180,E1 16463.509,E2 16463.509} C_VEL
LIN {X 0,Y 344.735,Z 1044.764,A -85,B 0,C 180,E1 16460.653,E2 16460.653} C_VEL
LIN {X 0,Y 344.79,Z 1038.485,A -85,B 0,C 180,E1 16457.759,E2 16457.759} C_VEL
LIN {X 0,Y 345.294,Z 1030.429,A -85,B 0,C 180,E1 16454.894,E2 16454.894} C_VEL
LIN {X 0,Y 346.271,Z 1020.883,A -85,B 0,C 180,E1 16452.177,E2 16452.177} C_VEL
LIN {X 0,Y 347.856,Z 1009.195,A -85,B 0,C 180,E1 16449.472,E2 16449.472} C_VEL
LIN {X 0,Y 349.77,Z 996.819,A -85,B 0,C 180,E1 16447.122,E2 16447.122} C_VEL
LIN {X 0,Y 352.02,Z 983.018,A -85,B 0,C 180,E1 16444.963,E2 16444.963} C_VEL
LIN {X 0,Y 354.548,Z 967.793,A -85,B 0,C 180,E1 16443.018,E2 16443.018} C_VEL
LIN {X 0,Y 357.036,Z 951.983,A -85,B 0,C 180,E1 16441.388,E2 16441.388} C_VEL
LIN {X 0,Y 359.416,Z 935.125,A -85,B 0,C 180,E1 16440.014,E2 16440.014} C_VEL
LIN {X 0,Y 361.521,Z 918.031,A -85,B 0,C 180,E1 16438.949,E2 16438.949} C_VEL
LIN {X 0,Y 363.28,Z 899.943,A -85,B 0,C 180,E1 16438.135,E2 16438.135} C_VEL
LIN {X 0,Y 364.397,Z 881.207,A -85,B 0,C 180,E1 16437.581,E2 16437.581} C_VEL
LIN {X 0,Y 368.727,Z 723.673,A -85,B 0,C 180,E1 16434.43,E2 16434.43} C_VEL
LIN {X 0,Y 365.795,Z 695.364,A -85,B 0,C 180,E1 16433.4,E2 16433.4} C_VEL
LIN {X 0,Y 369.634,Z 673.831,A -85,B 0,C 180,E1 16430.821,E2 16430.821} C_VEL
LIN {X 0,Y 365.251,Z 659.629,A -85,B 0,C 180,E1 16428.092,E2 16428.092} C_VEL
LIN {X 0,Y 360.226,Z 645.792,A -85,B 0,C 180,E1 16425.055,E2 16425.055} C_VEL
LIN {X 0,Y 355.157,Z 633.206,A -85,B 0,C 180,E1 16421.852,E2 16421.852} C_VEL
LIN {X 0,Y 351.063,Z 624.293,A -85,B 0,C 180,E1 16419.218,E2 16419.218} C_VEL
LIN {X 0,Y 347.602,Z 616.772,A -85,B 0,C 180,E1 16416.748,E2 16416.748} C_VEL
LIN {X 0,Y 345.928,Z 612.854,A -85,B 0,C 180,E1 16415.288,E2 16415.288} C_VEL
LIN {X 0,Y 345.905,Z 612.693,A -85,B 0,C 180,E1 16411.158,E2 16411.158} C_VEL
LIN {X 0,Y 345.916,Z 612.69,A -85,B 0,C 180,E1 16407.094,E2 16407.094} C_VEL
LIN {X 0,Y 345.92,Z 612.687,A -85,B 0,C 180,E1 16402.967,E2 16402.967} C_VEL
LIN {X 0,Y 345.912,Z 612.685,A -85,B 0,C 180,E1 16398.714,E2 16398.714} C_VEL
LIN {X 0,Y 345.913,Z 612.685,A -85,B 0,C 180,E1 16394.564,E2 16394.564} C_VEL
LIN {X 0,Y 345.908,Z 612.688,A -85,B 0,C 180,E1 16390.324,E2 16390.324} C_VEL
LIN {X 0,Y 345.908,Z 612.699,A -85,B 0,C 180,E1 16386.097,E2 16386.097} C_VEL
LIN {X 0,Y 345.905,Z 612.709,A -85,B 0,C 180,E1 16381.822,E2 16381.822} C_VEL
LIN {X 0,Y 345.908,Z 612.71,A -85,B 0,C 180,E1 16377.68,E2 16377.68} C_VEL
LIN {X 0,Y 345.909,Z 612.702,A -85,B 0,C 180,E1 16373.527,E2 16373.527} C_VEL
LIN {X 0,Y 345.91,Z 612.699,A -85,B 0,C 180,E1 16369.339,E2 16369.339} C_VEL
LIN {X 0,Y 345.908,Z 612.703,A -85,B 0,C 180,E1 16365.092,E2 16365.092} C_VEL
LIN {X 0,Y 345.913,Z 612.711,A -85,B 0,C 180,E1 16360.936,E2 16360.936} C_VEL
LIN {X 0,Y 345.983,Z 613.087,A -85,B 0,C 180,E1 16359.709,E2 16359.709} C_VEL
LIN {X 0,Y 349.405,Z 621.301,A -85,B 0,C 180,E1 16356.561,E2 16356.561} C_VEL
LIN {X 0,Y 353.303,Z 630.998,A -85,B 0,C 180,E1 16353.257,E2 16353.257} C_VEL
LIN {X 0,Y 357.373,Z 642.713,A -85,B 0,C 180,E1 16349.761,E2 16349.761} C_VEL
LIN {X 0,Y 361.089,Z 655.161,A -85,B 0,C 180,E1 16346.457,E2 16346.457} C_VEL
LIN {X 0,Y 364.177,Z 667.83,A -85,B 0,C 180,E1 16343.431,E2 16343.431} C_VEL
LIN {X 0,Y 360.853,Z 688.363,A -85,B 0,C 180,E1 16339.884,E2 16339.884} C_VEL
LIN {X 0,Y 358.197,Z 705.926,A -85,B 0,C 180,E1 16336.919,E2 16336.919} C_VEL
LIN {X 0,Y 359.158,Z 711.11,A -85,B 0,C 180,E1 16336.606,E2 16336.606} C_VEL
LIN {X 0,Y 364.784,Z 740.471,A -85,B 0,C 180,E1 16335.258,E2 16335.258} C_VEL
LIN {X 0,Y 365.008,Z 745.025,A -85,B 0,C 180,E1 16335.122,E2 16335.122} C_VEL
LIN {X 0,Y 361.972,Z 836.145,A -85,B 0,C 180,E1 16333.117,E2 16333.117} C_VEL
LIN {X 0,Y 361.089,Z 852.403,A -85,B 0,C 180,E1 16332.457,E2 16332.457} C_VEL
LIN {X 0,Y 359.9,Z 866.683,A -85,B 0,C 180,E1 16331.604,E2 16331.604} C_VEL
LIN {X 0,Y 358.181,Z 881.816,A -85,B 0,C 180,E1 16330.363,E2 16330.363} C_VEL
LIN {X 0,Y 356.326,Z 894.978,A -85,B 0,C 180,E1 16328.943,E2 16328.943} C_VEL
LIN {X 0,Y 354.359,Z 907.058,A -85,B 0,C 180,E1 16327.279,E2 16327.279} C_VEL
LIN {X 0,Y 352.4,Z 917.924,A -85,B 0,C 180,E1 16325.366,E2 16325.366} C_VEL
LIN {X 0,Y 350.517,Z 927.561,A -85,B 0,C 180,E1 16323.208,E2 16323.208} C_VEL
LIN {X 0,Y 348.868,Z 935.488,A -85,B 0,C 180,E1 16320.865,E2 16320.865} C_VEL
LIN {X 0,Y 347.637,Z 941.406,A -85,B 0,C 180,E1 16318.518,E2 16318.518} C_VEL
LIN {X 0,Y 346.658,Z 946.023,A -85,B 0,C 180,E1 16315.819,E2 16315.819} C_VEL
LIN {X 0,Y 346.105,Z 948.511,A -85,B 0,C 180,E1 16313.267,E2 16313.267} C_VEL
LIN {X 0,Y 345.826,Z 949.316,A -85,B 0,C 180,E1 16310.477,E2 16310.477} C_VEL
LIN {X 0,Y 345.814,Z 948.225,A -85,B 0,C 180,E1 16307.847,E2 16307.847} C_VEL
LIN {X 0,Y 346.069,Z 945.36,A -85,B 0,C 180,E1 16305.204,E2 16305.204} C_VEL
LIN {X 0,Y 346.658,Z 940.334,A -85,B 0,C 180,E1 16302.493,E2 16302.493} C_VEL
LIN {X 0,Y 347.509,Z 933.965,A -85,B 0,C 180,E1 16300.108,E2 16300.108} C_VEL
LIN {X 0,Y 348.726,Z 925.536,A -85,B 0,C 180,E1 16297.744,E2 16297.744} C_VEL
LIN {X 0,Y 350.181,Z 915.358,A -85,B 0,C 180,E1 16295.571,E2 16295.571} C_VEL
LIN {X 0,Y 351.64,Z 904.526,A -85,B 0,C 180,E1 16293.749,E2 16293.749} C_VEL
LIN {X 0,Y 353.245,Z 891.513,A -85,B 0,C 180,E1 16292.027,E2 16292.027} C_VEL
LIN {X 0,Y 354.708,Z 877.961,A -85,B 0,C 180,E1 16290.646,E2 16290.646} C_VEL
LIN {X 0,Y 355.98,Z 863.521,A -85,B 0,C 180,E1 16289.517,E2 16289.517} C_VEL
LIN {X 0,Y 357.013,Z 847.067,A -85,B 0,C 180,E1 16288.602,E2 16288.602} C_VEL
LIN {X 0,Y 357.598,Z 831.167,A -85,B 0,C 180,E1 16288.042,E2 16288.042} C_VEL
LIN {X 0,Y 359.973,Z 740.884,A -85,B 0,C 180,E1 16286.143,E2 16286.143} C_VEL
LIN {X 0,Y 359.336,Z 735.558,A -85,B 0,C 180,E1 16285.975,E2 16285.975} C_VEL
LIN {X 0,Y 356.593,Z 728.672,A -85,B 0,C 180,E1 16285.606,E2 16285.606} C_VEL
LIN {X 0,Y 349.334,Z 715.597,A -85,B 0,C 180,E1 16284.722,E2 16284.722} C_VEL
LIN {X 0,Y 347.395,Z 709.374,A -85,B 0,C 180,E1 16284.417,E2 16284.417} C_VEL
LIN {X 0,Y 346.939,Z 706.033,A -85,B 0,C 180,E1 16284.252,E2 16284.252} C_VEL
LIN {X 0,Y 350.462,Z 678.347,A -85,B 0,C 180,E1 16279.645,E2 16279.645} C_VEL
LIN {X 0,Y 352.496,Z 662.984,A -85,B 0,C 180,E1 16277.051,E2 16277.051} C_VEL
LIN {X 0,Y 348.267,Z 646.446,A -85,B 0,C 180,E1 16273.487,E2 16273.487} C_VEL
LIN {X 0,Y 343.659,Z 630.746,A -85,B 0,C 180,E1 16269.832,E2 16269.832} C_VEL
LIN {X 0,Y 338.778,Z 616.273,A -85,B 0,C 180,E1 16266.196,E2 16266.196} C_VEL
LIN {X 0,Y 337.988,Z 613.769,A -85,B 0,C 180,E1 16265.44,E2 16265.44} C_VEL
LIN {X 0,Y 337.975,Z 613.652,A -85,B 0,C 180,E1 16261.127,E2 16261.127} C_VEL
LIN {X 0,Y 337.976,Z 613.658,A -85,B 0,C 180,E1 16256.817,E2 16256.817} C_VEL
LIN {X 0,Y 337.976,Z 613.678,A -85,B 0,C 180,E1 16252.665,E2 16252.665} C_VEL
LIN {X 0,Y 337.976,Z 613.684,A -85,B 0,C 180,E1 16248.459,E2 16248.459} C_VEL
LIN {X 0,Y 337.979,Z 613.697,A -85,B 0,C 180,E1 16244.28,E2 16244.28} C_VEL
LIN {X 0,Y 337.981,Z 613.668,A -85,B 0,C 180,E1 16239.938,E2 16239.938} C_VEL
LIN {X 0,Y 337.98,Z 613.68,A -85,B 0,C 180,E1 16235.648,E2 16235.648} C_VEL
LIN {X 0,Y 337.987,Z 613.686,A -85,B 0,C 180,E1 16231.377,E2 16231.377} C_VEL
LIN {X 0,Y 337.991,Z 613.661,A -85,B 0,C 180,E1 16227.071,E2 16227.071} C_VEL
LIN {X 0,Y 338,Z 613.694,A -85,B 0,C 180,E1 16222.617,E2 16222.617} C_VEL
LIN {X 0,Y 337.981,Z 613.655,A -85,B 0,C 180,E1 16218.262,E2 16218.262} C_VEL
LIN {X 0,Y 337.984,Z 613.695,A -85,B 0,C 180,E1 16213.991,E2 16213.991} C_VEL
LIN {X 0,Y 337.969,Z 613.657,A -85,B 0,C 180,E1 16209.709,E2 16209.709} C_VEL
LIN {X 0,Y 337.977,Z 613.693,A -85,B 0,C 180,E1 16205.603,E2 16205.603} C_VEL
LIN {X 0,Y 337.966,Z 613.66,A -85,B 0,C 180,E1 16201.357,E2 16201.357} C_VEL
LIN {X 0,Y 337.965,Z 613.697,A -85,B 0,C 180,E1 16197.117,E2 16197.117} C_VEL
LIN {X 0,Y 337.956,Z 613.661,A -85,B 0,C 180,E1 16192.862,E2 16192.862} C_VEL
LIN {X 0,Y 337.956,Z 613.699,A -85,B 0,C 180,E1 16188.567,E2 16188.567} C_VEL
LIN {X 0,Y 337.951,Z 613.679,A -85,B 0,C 180,E1 16184.382,E2 16184.382} C_VEL
LIN {X 0,Y 337.95,Z 613.679,A -85,B 0,C 180,E1 16180.109,E2 16180.109} C_VEL
LIN {X 0,Y 337.949,Z 613.701,A -85,B 0,C 180,E1 16175.903,E2 16175.903} C_VEL
LIN {X 0,Y 337.949,Z 613.701,A -85,B 0,C 180,E1 16171.554,E2 16171.554} C_VEL
LIN {X 0,Y 337.947,Z 613.7,A -85,B 0,C 180,E1 16167.421,E2 16167.421} C_VEL
LIN {X 0,Y 337.949,Z 613.705,A -85,B 0,C 180,E1 16163.088,E2 16163.088} C_VEL
LIN {X 0,Y 338.008,Z 613.954,A -85,B 0,C 180,E1 16159.845,E2 16159.845} C_VEL
LIN {X 0,Y 344.27,Z 630.154,A -85,B 0,C 180,E1 16156.274,E2 16156.274} C_VEL
LIN {X 0,Y 350.577,Z 647.671,A -85,B 0,C 180,E1 16152.864,E2 16152.864} C_VEL
LIN {X 0,Y 357.09,Z 667.46,A -85,B 0,C 180,E1 16149.394,E2 16149.394} C_VEL
LIN {X 0,Y 358.346,Z 672.271,A -85,B 0,C 180,E1 16148.624,E2 16148.624} C_VEL
LIN {X 0,Y 354.889,Z 695.345,A -85,B 0,C 180,E1 16145.946,E2 16145.946} C_VEL
LIN {X 0,Y 357.807,Z 726.969,A -85,B 0,C 180,E1 16144.994,E2 16144.994} C_VEL
LIN {X 0,Y 353.752,Z 887.562,A -85,B 0,C 180,E1 16141.801,E2 16141.801} C_VEL
LIN {X 0,Y 352.559,Z 905.98,A -85,B 0,C 180,E1 16141.158,E2 16141.158} C_VEL
LIN {X 0,Y 350.853,Z 923.816,A -85,B 0,C 180,E1 16140.246,E2 16140.246} C_VEL
LIN {X 0,Y 348.914,Z 940.777,A -85,B 0,C 180,E1 16139.071,E2 16139.071} C_VEL
LIN {X 0,Y 346.726,Z 957.604,A -85,B 0,C 180,E1 16137.571,E2 16137.571} C_VEL
LIN {X 0,Y 344.468,Z 973.344,A -85,B 0,C 180,E1 16135.811,E2 16135.811} C_VEL
LIN {X 0,Y 342.327,Z 988.114,A -85,B 0,C 180,E1 16133.771,E2 16133.771} C_VEL
LIN {X 0,Y 340.442,Z 1001.312,A -85,B 0,C 180,E1 16131.538,E2 16131.538} C_VEL
LIN {X 0,Y 338.896,Z 1013.109,A -85,B 0,C 180,E1 16129.117,E2 16129.117} C_VEL
LIN {X 0,Y 337.724,Z 1023.844,A -85,B 0,C 180,E1 16126.418,E2 16126.418} C_VEL
LIN {X 0,Y 337.054,Z 1033.007,A -85,B 0,C 180,E1 16123.554,E2 16123.554} C_VEL
LIN {X 0,Y 336.831,Z 1040.4,A -85,B 0,C 180,E1 16120.606,E2 16120.606} C_VEL
LIN {X 0,Y 336.968,Z 1045.911,A -85,B 0,C 180,E1 16117.671,E2 16117.671} C_VEL
LIN {X 0,Y 337.25,Z 1049.643,A -85,B 0,C 180,E1 16114.762,E2 16114.762} C_VEL
LIN {X 0,Y 337.487,Z 1051.68,A -85,B 0,C 180,E1 16111.868,E2 16111.868} C_VEL
LIN {X 0,Y 337.513,Z 1052.082,A -85,B 0,C 180,E1 16109.152,E2 16109.152} C_VEL
LIN {X 0,Y 337.315,Z 1051.034,A -85,B 0,C 180,E1 16106.431,E2 16106.431} C_VEL
LIN {X 0,Y 336.995,Z 1048.316,A -85,B 0,C 180,E1 16103.527,E2 16103.527} C_VEL
LIN {X 0,Y 336.754,Z 1043.606,A -85,B 0,C 180,E1 16100.429,E2 16100.429} C_VEL
LIN {X 0,Y 336.829,Z 1037.379,A -85,B 0,C 180,E1 16097.485,E2 16097.485} C_VEL
LIN {X 0,Y 337.386,Z 1029.288,A -85,B 0,C 180,E1 16094.531,E2 16094.531} C_VEL
LIN {X 0,Y 338.452,Z 1019.776,A -85,B 0,C 180,E1 16091.751,E2 16091.751} C_VEL
LIN {X 0,Y 340.156,Z 1008.099,A -85,B 0,C 180,E1 16088.985,E2 16088.985} C_VEL
LIN {X 0,Y 342.249,Z 995.452,A -85,B 0,C 180,E1 16086.539,E2 16086.539} C_VEL
LIN {X 0,Y 344.699,Z 981.341,A -85,B 0,C 180,E1 16084.301,E2 16084.301} C_VEL
LIN {X 0,Y 347.305,Z 966.521,A -85,B 0,C 180,E1 16082.387,E2 16082.387} C_VEL
LIN {X 0,Y 349.891,Z 950.843,A -85,B 0,C 180,E1 16080.748,E2 16080.748} C_VEL
LIN {X 0,Y 352.355,Z 934.338,A -85,B 0,C 180,E1 16079.379,E2 16079.379} C_VEL
LIN {X 0,Y 354.606,Z 916.849,A -85,B 0,C 180,E1 16078.274,E2 16078.274} C_VEL
LIN {X 0,Y 356.431,Z 898.941,A -85,B 0,C 180,E1 16077.46,E2 16077.46} C_VEL
LIN {X 0,Y 357.586,Z 880.162,A -85,B 0,C 180,E1 16076.899,E2 16076.899} C_VEL
LIN {X 0,Y 362.097,Z 724.56,A -85,B 0,C 180,E1 16073.736,E2 16073.736} C_VEL
LIN {X 0,Y 359.138,Z 695.472,A -85,B 0,C 180,E1 16072.639,E2 16072.639} C_VEL
LIN {X 0,Y 362.597,Z 676.487,A -85,B 0,C 180,E1 16070.295,E2 16070.295} C_VEL
LIN {X 0,Y 358.204,Z 662.288,A -85,B 0,C 180,E1 16067.468,E2 16067.468} C_VEL
LIN {X 0,Y 353.276,Z 648.657,A -85,B 0,C 180,E1 16064.352,E2 16064.352} C_VEL
LIN {X 0,Y 348.496,Z 637.063,A -85,B 0,C 180,E1 16061.263,E2 16061.263} C_VEL
LIN {X 0,Y 345.105,Z 629.411,A -85,B 0,C 180,E1 16058.954,E2 16058.954} C_VEL
LIN {X 0,Y 341.681,Z 621.995,A -85,B 0,C 180,E1 16056.444,E2 16056.444} C_VEL
LIN {X 0,Y 339.611,Z 617.666,A -85,B 0,C 180,E1 16054.831,E2 16054.831} C_VEL
LIN {X 0,Y 337.989,Z 613.837,A -85,B 0,C 180,E1 16053.231,E2 16053.231} C_VEL
LIN {X 0,Y 337.969,Z 613.689,A -85,B 0,C 180,E1 16049.024,E2 16049.024} C_VEL
LIN {X 0,Y 337.959,Z 613.687,A -85,B 0,C 180,E1 16044.733,E2 16044.733} C_VEL
LIN {X 0,Y 337.962,Z 613.692,A -85,B 0,C 180,E1 16040.613,E2 16040.613} C_VEL
LIN {X 0,Y 337.966,Z 613.699,A -85,B 0,C 180,E1 16036.499,E2 16036.499} C_VEL
LIN {X 0,Y 337.965,Z 613.697,A -85,B 0,C 180,E1 16032.298,E2 16032.298} C_VEL
LIN {X 0,Y 337.96,Z 613.685,A -85,B 0,C 180,E1 16027.993,E2 16027.993} C_VEL
LIN {X 0,Y 337.955,Z 613.678,A -85,B 0,C 180,E1 16023.732,E2 16023.732} C_VEL
LIN {X 0,Y 337.956,Z 613.675,A -85,B 0,C 180,E1 16019.491,E2 16019.491} C_VEL
LIN {X 0,Y 337.956,Z 613.676,A -85,B 0,C 180,E1 16015.248,E2 16015.248} C_VEL
LIN {X 0,Y 337.957,Z 613.677,A -85,B 0,C 180,E1 16010.978,E2 16010.978} C_VEL
LIN {X 0,Y 337.958,Z 613.679,A -85,B 0,C 180,E1 16006.657,E2 16006.657} C_VEL
LIN {X 0,Y 337.964,Z 613.688,A -85,B 0,C 180,E1 16002.294,E2 16002.294} C_VEL
LIN {X 0,Y 338.037,Z 614.037,A -85,B 0,C 180,E1 16001.707,E2 16001.707} C_VEL
LIN {X 0,Y 340.287,Z 619.586,A -85,B 0,C 180,E1 15999.354,E2 15999.354} C_VEL
LIN {X 0,Y 343.118,Z 625.966,A -85,B 0,C 180,E1 15996.834,E2 15996.834} C_VEL
LIN {X 0,Y 346.907,Z 635.651,A -85,B 0,C 180,E1 15993.465,E2 15993.465} C_VEL
LIN {X 0,Y 350.877,Z 647.348,A -85,B 0,C 180,E1 15989.898,E2 15989.898} C_VEL
LIN {X 0,Y 354.382,Z 659.419,A -85,B 0,C 180,E1 15986.62,E2 15986.62} C_VEL
LIN {X 0,Y 357.185,Z 671.336,A -85,B 0,C 180,E1 15983.725,E2 15983.725} C_VEL
LIN {X 0,Y 352.538,Z 698.075,A -85,B 0,C 180,E1 15979.068,E2 15979.068} C_VEL
LIN {X 0,Y 351.342,Z 706.069,A -85,B 0,C 180,E1 15977.724,E2 15977.724} C_VEL
LIN {X 0,Y 355.081,Z 724.64,A -85,B 0,C 180,E1 15976.739,E2 15976.739} C_VEL
LIN {X 0,Y 358.44,Z 744.446,A -85,B 0,C 180,E1 15975.856,E2 15975.856} C_VEL
LIN {X 0,Y 355.203,Z 836.781,A -85,B 0,C 180,E1 15973.79,E2 15973.79} C_VEL
LIN {X 0,Y 354.273,Z 853.069,A -85,B 0,C 180,E1 15973.119,E2 15973.119} C_VEL
LIN {X 0,Y 353.047,Z 867.159,A -85,B 0,C 180,E1 15972.269,E2 15972.269} C_VEL
LIN {X 0,Y 351.268,Z 882.091,A -85,B 0,C 180,E1 15971.035,E2 15971.035} C_VEL
LIN {X 0,Y 349.395,Z 894.917,A -85,B 0,C 180,E1 15969.654,E2 15969.654} C_VEL
LIN {X 0,Y 347.15,Z 907.959,A -85,B 0,C 180,E1 15967.841,E2 15967.841} C_VEL
LIN {X 0,Y 345.191,Z 918.26,A -85,B 0,C 180,E1 15966.015,E2 15966.015} C_VEL
LIN {X 0,Y 343.153,Z 928.02,A -85,B 0,C 180,E1 15963.816,E2 15963.816} C_VEL
LIN {X 0,Y 341.444,Z 935.734,A -85,B 0,C 180,E1 15961.554,E2 15961.554} C_VEL
LIN {X 0,Y 339.998,Z 942.163,A -85,B 0,C 180,E1 15959.027,E2 15959.027} C_VEL
LIN {X 0,Y 338.96,Z 946.677,A -85,B 0,C 180,E1 15956.45,E2 15956.45} C_VEL
